# B&R Automation Studio project CombinedLinenSoiledA9KAN (part 2)

#### picu.ab
```automation-basic
PROGRAM _CYCLIC

;Sequence 24 - Primary Incline Conveyor 1 D[900 + mySeq]

;Note - Not a real sequence and not shown

;-----------------------------------------
;Revision 1.00 17/04/2007 D.J. First Issue
;-----------------------------------------

mySeq = 31
myIO = 172
myX20IO	= 23
myBufferBag = 841
myRelLine	= 65
myLine = 82 ; Line used to track bags
myZone	= 4

myLastBag = Line[myLine].LastBag
myFirstBag = Line[myLine].FirstBag
myRelBag = Line[myRelLine].LastBag

I_PaddleInPosition		= X[myIO].X01
I_BagReleasedSep		= X[myIO].X02
I_BagAtSep              = X[myIO].X03
I_ArriveIncline			= X[myIO].X04

O_RunMotor 				= FALSE
O_OpenSeparator			= FALSE

Alarm[mySeq].Name 	= 0
Alarm[mySeq].Bag	= myFirstBag
Alarm[mySeq].Beacon	= TRUE
Alarm[mySeq].Extra	= 0
Alarm[mySeq].Time	= 3000

;Setup Sequence
;-----------------------
STEP = D[900 + mySeq]
;Setup Pulse contact
PLS = (STEP <> LASTSTEP)
LASTSTEP = STEP

;If no bags on the buffers then stop the motor
NoBags = (Bag[myBufferBag].Cat = 0) AND (Bag[myFirstBag].Cat = 0)
TON_10ms(NoBags,10,StopIncline,StopInclineET)

O_RunMotor = (Line[myRelLine].Clear AND NOT Line[myRelLine].TripFault AND NOT StopIncline AND NOT Std.HaltSysZone[myZone] AND (STEP <> 2) AND (STEP <> 0))
IF (STEP = 0) THEN

ENDIF

;Run Incline until paddle in position
TON_10ms(I_BagAtSep,250,SettledInSep,SettledInSepET)
TON_10ms((Bag[myBufferBag].Cat > 0) AND NOT Std.HaltSysZone[myZone],300,SettledAtSep,SettledAtSepET)
IF (STEP = 1) THEN
	IF (I_PaddleInPosition AND O_RunMotor AND SettledAtSep AND (Bag[myLastBag].Cat = 0) AND (Bag[myBufferBag].Cat > 0)) THEN
		D[900 + mySeq] = 2
	ENDIF
ENDIF

;Release Bag into incline
IF (STEP = 2) THEN
	IF SettledInSep THEN
		BagArrived = TRUE
	ENDIF
	O_OpenSeparator	= (Bag[myLastBag].Cat = 0) AND NOT BagArrived

	IF I_ArriveIncline THEN
		IF ((Bag[myBufferBag].Cat > 0) AND (Bag[myLastBag].Cat = 0)) THEN
			Bag[myLastBag] = Bag[myBufferBag]
			Bag[myBufferBag] = Bag[0]
		ENDIF
		D[900 + mySeq] = 3
	ENDIF
	IF (Bag[myLastBag].Cat > 0) THEN
		Alarm[mySeq].Name = almBagDataError
		Alarm[mySeq].Time = 0
		Alarm[mySeq].Bag = myLastBag
	ELSE IF (Bag[myBufferBag].Cat > 0) AND NOT I_BagAtSep THEN
		Alarm[mySeq].Name = almSwitchFault
		Alarm[mySeq].Bag = myBufferBag
	ELSE
		Alarm[mySeq].Name = almBagNotReleased
		Alarm[mySeq].Bag = myBufferBag
	ENDIF
ELSE
	BagArrived = FALSE
ENDIF

;Check not stpped on paddle
IF (STEP = 3) THEN
	IF NOT I_PaddleInPosition THEN
		D[900 + mySeq] = 1
	ENDIF
ENDIF

;Move data from incline..
IF Line[myRelLine].Trip AND (Bag[myFirstBag].Cat > 0) AND (Bag[myRelBag].Cat = 0)  THEN ; Trip includes debounce
	Bag[myRelBag] = Bag[myFirstBag]
	Bag[myFirstBag] = Bag[0]
ENDIF

;Alarms
TimerAlarm.IN 		= NOT PLS AND (Alarm[mySeq].Name > 0)
TimerAlarm.PT 		= Alarm[mySeq].Time
TimerAlarm FUB TON_10ms()
Alarm[mySeq].On 	= TimerAlarm.Q
Alarm[mySeq].ET 	= TimerAlarm.ET
Alarm[mySeq].Zone 	= myZone

Y[myX20IO].Y02 	= O_RunMotor
Y[myIO].Y06 	= O_OpenSeparator AND NOT OpenSep
END_PROGRAM
```

### Program Logical/Reference/32_picd3 (IEC) - *PICD3 Incline Down Full bags

#### picd.var
```iecst
VAR
	TransitWindowClosedET : TIME;
	TransitWindowClosed : BOOL;
	TimerAlarm : TON_10ms;
	StopInclineET : TIME;
	StopIncline : BOOL;
	STEP : UINT;
	SettledAtSepET : UDINT;
	SettledAtSep : BOOL;
	ReleasedToInclineET : TIME;
	ReleasedToIncline : BOOL;
END_VAR
VAR RETAIN
	PLS : BOOL;
END_VAR
VAR
	O_RunMotor : BOOL;
	O_OpenSeparator : BOOL;
	NoBags : BOOL;
	myZone : INT;
	myX20IO : UINT;
	mySeq : UINT;
	myRelLine : UINT;
	myRelBag : UINT;
	myLine : UINT;
	myLastBag : UINT;
	myIO : UINT;
	myFirstBag : UINT;
	myBufferBag : UINT;
END_VAR
VAR RETAIN
	LASTSTEP : UINT;
END_VAR
VAR
	I_TrolleyOutAtBott : BOOL;
	I_TrolleyOnIncline : BOOL;
	I_PaddleInPosition : BOOL;
	I_OutgoingFull : BOOL;
	I_BagInSep : BOOL;
	I_BagAtSep : BOOL;
	I_ArriveIncline : BOOL;
	BagReleasedSep : BOOL;
	BagReleased : BOOL;
	BagArriveIncline : BOOL;
	SettledInSep : BOOL;
	SettledInSepET : UDINT;
	BagArrived : BOOL;
END_VAR
```

#### picd.ab
```automation-basic
PROGRAM _CYCLIC

;Sequence 24 - Primary Incline Conveyor 1 D[900 + mySeq]

;Note - Not a real sequence and not shown

;-----------------------------------------
;Revision 1.00 17/04/2007 D.J. First Issue
;-----------------------------------------

mySeq = 32
myIO = 173
myX20IO	= 33
myBufferBag = 891
myRelLine	= 68
myLine = 83 ; Line used to track bags
myZone	= 1

myLastBag = Line[myLine].LastBag
myFirstBag = Line[myLine].FirstBag
myRelBag = Line[myRelLine].LastBag

I_PaddleInPosition		= X[myIO].X01
I_BagInSep				= X[myIO].X02
I_BagAtSep              = X[myIO].X03
I_ArriveIncline			= X[myIO].X04

O_RunMotor 				= FALSE
O_OpenSeparator			= FALSE

Alarm[mySeq].Name 	= 0
Alarm[mySeq].Bag	= myFirstBag
Alarm[mySeq].Beacon	= TRUE
Alarm[mySeq].Extra	= 0
Alarm[mySeq].Time	= 3000

;Setup Sequence
;-----------------------
STEP = D[900 + mySeq]
;Setup Pulse contact
PLS = (STEP <> LASTSTEP)
LASTSTEP = STEP

;If no bags on the buffers then stop the motor
;NoBags = (Bag[myBufferBag].Cat = 0) AND (Bag[myFirstBag].Cat = 0)
NoBags = (((Bag[myFirstBag].Cat = 0) OR ((STEP = 1) AND Bag[myBufferBag].Cat > 0))  AND ((STEP = 1) AND I_PaddleInPosition))
IF NoBags THEN
	StopIncline = TRUE
ELSE IF (STEP <> 1) THEN
	StopIncline = FALSE
ENDIF

O_RunMotor = (Line[myRelLine].Clear AND NOT Line[myRelLine].TripFault AND NOT Std.HaltSysZone[myZone] AND (STEP <> 2) AND (STEP <> 0))
IF (STEP = 0) THEN

ENDIF

;Run Incline until paddle in position
TON_10ms(I_BagAtSep,25,SettledAtSep,SettledAtSepET)	;75
IF (STEP = 1) THEN
	IF ((I_PaddleInPosition OR StopIncline) AND O_RunMotor AND SettledAtSep AND (Bag[myLastBag].Cat = 0) AND (Bag[myBufferBag].Cat > 0) AND NOT I_BagInSep) THEN
		D[900 + mySeq] = 2
	ENDIF
	IF I_BagInSep THEN
		Alarm[mySeq].Name = almSwitchFault
	ENDIF
ENDIF

;Release Bag into incline

TON_10ms(I_BagInSep,25,SettledInSep,SettledInSepET)	;150
IF (STEP = 2) THEN

	IF SettledInSep THEN
		BagArrived = TRUE
	ENDIF
	O_OpenSeparator	= (Bag[myLastBag].Cat = 0) AND NOT BagArrived
	IF I_ArriveIncline THEN
		IF ((Bag[myBufferBag].Cat > 0) AND (Bag[myLastBag].Cat = 0)) THEN
			Bag[myLastBag] = Bag[myBufferBag]
			Bag[myBufferBag] = Bag[0]
		ENDIF
		D[900 + mySeq] = 3
	ENDIF
	IF (Bag[myLastBag].Cat > 0) THEN
		Alarm[mySeq].Name = almBagDataError
		Alarm[mySeq].Time = 0
		Alarm[mySeq].Bag = myLastBag
	ELSE
		Alarm[mySeq].Name = almBagNotReleased
		Alarm[mySeq].Bag = myBufferBag
	ENDIF
ELSE
	BagArrived = FALSE
ENDIF

;Check not stpped on paddle
IF (STEP = 3) THEN
	IF NOT I_PaddleInPosition THEN
		D[900 + mySeq] = 1
	ENDIF
ENDIF

;Move data from incline..
IF Line[myRelLine].Trip AND (Bag[myFirstBag].Cat > 0) AND (Bag[myRelBag].Cat = 0)  THEN ; Trip includes debounce
	Bag[myRelBag] = Bag[myFirstBag]
	Bag[myFirstBag] = Bag[0]
ENDIF

;Alarms
TimerAlarm.IN 		= NOT PLS AND (Alarm[mySeq].Name > 0)
TimerAlarm.PT 		= Alarm[mySeq].Time
TimerAlarm FUB TON_10ms()
Alarm[mySeq].On 	= TimerAlarm.Q
Alarm[mySeq].ET 	= TimerAlarm.ET
Alarm[mySeq].Zone 	= myZone

Y[myX20IO].Y01 	= O_RunMotor AND NOT StopIncline
Y[myIO].Y06 	= O_OpenSeparator
END_PROGRAM
```

### Program Logical/Reference/33_picd4 (IEC) - *PICD4 Incline Down Full bags

#### picd.ab
```automation-basic
PROGRAM _CYCLIC

;Sequence 24 - Primary Incline Conveyor 1 D[900 + mySeq]

;Note - Not a real sequence and not shown

;-----------------------------------------
;Revision 1.00 17/04/2007 D.J. First Issue
;-----------------------------------------

mySeq = 33
myIC = 4
myIO = 174
myX20IO	= 33
myBufferBag = 907
myRelLine	= 69
myLine = 84 ; Line used to track bags
myZone	= 1

myLastBag = Line[myLine].LastBag
myFirstBag = Line[myLine].FirstBag
myRelBag = Line[myRelLine].LastBag

I_PaddleInPosition		= X[myIO].X01
I_BagInSep				= X[myIO].X02
I_BagAtSep              = X[myIO].X03
I_ArriveIncline			= X[myIO].X04

O_RunMotor 				= FALSE
O_OpenSeparator			= FALSE
Enable.IC[myIC]			= FALSE

Alarm[mySeq].Name 	= 0
Alarm[mySeq].Bag	= myFirstBag
Alarm[mySeq].Beacon	= TRUE
Alarm[mySeq].Extra	= 0
Alarm[mySeq].Time	= 3000

;Setup Sequence
;-----------------------
STEP = D[900 + mySeq]
;Setup Pulse contact
PLS = (STEP <> LASTSTEP)
LASTSTEP = STEP

;If no bags on the buffers then stop the motor
NoBags = (((Bag[myFirstBag].Cat = 0) OR ((STEP = 1) AND Bag[myBufferBag].Cat > 0))  AND ((STEP = 1) AND I_PaddleInPosition))
IF NoBags THEN
	StopIncline = TRUE
ELSE IF (STEP <> 1) THEN
	StopIncline = FALSE
ENDIF

O_RunMotor = (Line[myRelLine].Clear AND NOT Line[myRelLine].TripFault AND NOT Std.HaltSysZone[myZone] AND (STEP <> 2) AND (STEP <> 0))
IF (STEP = 0) THEN

ENDIF

;Run Incline until paddle in position
TON_10ms(I_BagAtSep,25,SettledAtSep,SettledAtSepET)	;75
IF (STEP = 1) THEN
	IF ((I_PaddleInPosition OR StopIncline) AND O_RunMotor AND SettledAtSep AND (Bag[myLastBag].Cat = 0) AND (Bag[myBufferBag].Cat > 0) AND NOT I_BagInSep) THEN
		D[900 + mySeq] = 2
	ENDIF
	IF I_BagInSep THEN
		Alarm[mySeq].Name = almSwitchFault
	ENDIF
ENDIF

;Release Bag into incline

TON_10ms(I_BagInSep,150,SettledInSep,SettledInSepET)
IF (STEP = 2) THEN
	IF SettledInSep THEN
		BagArrived = TRUE
	ENDIF
	O_OpenSeparator	= (Bag[myLastBag].Cat = 0) AND NOT BagArrived
	IF I_ArriveIncline THEN
		IF ((Bag[myBufferBag].Cat > 0) AND (Bag[myLastBag].Cat = 0)) THEN
			Bag[myLastBag] = Bag[myBufferBag]
			Bag[myBufferBag] = Bag[0]
		ENDIF
		D[900 + mySeq] = 3
	ENDIF
	IF (Bag[myLastBag].Cat > 0) THEN
		Alarm[mySeq].Name = almBagDataError
		Alarm[mySeq].Time = 0
		Alarm[mySeq].Bag = myLastBag
	ELSE
		Alarm[mySeq].Name = almBagNotReleased
		Alarm[mySeq].Bag = myBufferBag
	ENDIF
ELSE
	BagArrived = FALSE
ENDIF

;Check not stpped on paddle
IF (STEP = 3) THEN
	IF NOT I_PaddleInPosition THEN
		D[900 + mySeq] = 1
	ENDIF
ENDIF

;Move data from incline..
IF Line[myRelLine].Trip AND (Bag[myFirstBag].Cat > 0) AND (Bag[myRelBag].Cat = 0)  THEN ; Trip includes debounce
	Bag[myRelBag] = Bag[myFirstBag]
	Bag[myFirstBag] = Bag[0]
ENDIF

;Alarms
TimerAlarm.IN 		= NOT PLS AND (Alarm[mySeq].Name > 0)
TimerAlarm.PT 		= Alarm[mySeq].Time
TimerAlarm FUB TON_10ms()
Alarm[mySeq].On 	= TimerAlarm.Q
Alarm[mySeq].ET 	= TimerAlarm.ET
Alarm[mySeq].Zone 	= myZone
Y[myX20IO].Y02 	= O_RunMotor AND NOT StopIncline
Y[myIO].Y06 	= O_OpenSeparator
END_PROGRAM
```

### Program Logical/Reference/35_picu6 (IEC) - *PICU6 Incline up Empty trolleys - Special not outgoing buffer

#### picu.var
```iecst
VAR RETAIN
	STEP : UINT;
	PLS : BOOL;
	LASTSTEP : UINT;
END_VAR
VAR
	O_RunMotor : BOOL;
	I_OutgoingFull : BOOL;
	O_OpenSeparator : BOOL;
	ReleasedToIncline : BOOL;
	ReleasedToInclineET : TIME;
	OutgoingFull : BOOL;
	OutgoingFullET : TIME;
	NoBags : BOOL;
	StopInclineET : TIME;
	StopIncline : BOOL;
	I_PaddleInPosition : BOOL;
	BagArriveIncline : BOOL;
	I_ArriveIncline : BOOL;
	TransitWindowClosedET : TIME;
	TransitWindowClosed : BOOL;
	BagReleasedSep : BOOL;
	I_BagAtSep : BOOL;
	I_LoadingInPosition : BOOL;
	TrackInPosET : TIME;
	TrackInPos : BOOL;
	mySeq : UINT;
	I_BagArriveIncline : BOOL;
	myIO : UINT;
	I_BagAtTopIncline : BOOL;
	I_BagReleased : BOOL;
	myIC : UINT;
	SettledSep : BOOL;
	SettledSepET : UDINT;
	myZone : INT;
	I_BagInSep : BOOL;
	SettledInSep : BOOL;
	SettledInSepET : UDINT;
	BagInSep : BOOL;
END_VAR
```

#### picu.ab
```automation-basic
PROGRAM _CYCLIC
	(* cyclic program *)

;Sequence 30 - Primary Incline Conveyor 4 D[900 + mySeq]
;Special incline - Only use 1 bag at time to store as buffer.
;-----------------------------------------
;Revision 1.00 17/04/2007 D.J. First Issue
;-----------------------------------------
mySeq 	= 35
myIO	= 176
myIC 	= 6
myZone	= 0

I_PaddleInPosition		= X[myIO].X01
I_BagAtSep              = X[myIO].X03
I_BagArriveIncline		= X[myIO].X04
I_BagInSep				= X[myIO].X02
I_BagReleased			= X[myIO].X05

O_RunMotor 				= FALSE
O_OpenSeparator			= FALSE
RequestRel.IC[myIC]		= FALSE

;Setup Sequence
;-----------------------
STEP = D[900 + mySeq]
;Setup Pulse contact
PLS = (STEP <> LASTSTEP)
LASTSTEP = STEP

IF (STEP = 0) THEN
;	D[900 + mySeq] = 1
ENDIF

;Run Incline until paddle in position
IF (STEP = 1) THEN
	O_RunMotor = TRUE
	IF I_PaddleInPosition AND NOT I_BagAtTopIncline THEN
		D[900 + mySeq] = 2
	ELSE IF I_BagAtTopIncline THEN
		Alarm[mySeq].Name = almSwitchFault
	ENDIF
ENDIF

;Step 2 wait for trolley at sep
TON_10ms(I_BagAtSep,200,SettledSep,SettledSepET)
	IF (STEP = 2) THEN
		IF SettledSep THEN
		D[900 + mySeq] = 3
	ENDIF
ENDIF

;Open Separator 1.5 seconds
TON_10ms(I_BagInSep,150,SettledInSep,SettledInSepET)
IF (STEP = 3) THEN
	IF SettledInSep THEN
		BagInSep = TRUE
	ENDIF
	O_OpenSeparator = NOT BagInSep
	IF I_BagArriveIncline THEN
		D[900 + mySeq] = 4
	ENDIF
	IF NOT Std.HaltSysZone[myZone] THEN
		Alarm[mySeq].Name = almBagNotArrived
	ENDIF
ELSE
	BagInSep = FALSE
ENDIF

;Step 4 Run incline until trolley is at the top
IF (STEP = 4) THEN
;	O_RunMotor = NOT EnableRel.IC[myIC]
;	IF I_BagAtTopIncline THEN
	IF NOT EnableRel.IC[myIC] THEN
		D[900 + mySeq] = 5
	ENDIF
;	ENDIF
;	IF EnableRel.IC[myIC] THEN
;		Alarm[mySeq].Name = almGeneralSequence
;	ENDIF
ENDIF

;Step 5 RequestRel
IF (STEP = 5) THEN
	RequestRel.IC[myIC] = NOT I_BagReleased
	IF EnableRel.IC[myIC] THEN
		D[900 + mySeq] = 6
	ENDIF
	IF  I_BagReleased AND NOT Std.HaltSysZone[myZone] THEN
		Alarm[mySeq].Name = almSwitchFault
	ENDIF
ENDIF

;Step 6 Run To Release trolley
IF (STEP = 6) THEN
	O_RunMotor = TRUE
	IF (I_BagReleased OR NOT EnableRel.IC[myIC]) THEN
		D[900 + mySeq] = 7
	ENDIF

ENDIF

;Check not stpped on paddle
IF (STEP = 7) THEN
	O_RunMotor = TRUE
	IF NOT I_PaddleInPosition THEN
		D[900 + mySeq] = 1
	ENDIF
ENDIF

Y[34].Y01		= O_RunMotor
Y[myIO].Y06 	= O_OpenSeparator
END_PROGRAM
```

### Program Logical/Reference/37_picu8 (IEC) - *PICU8 Incline up Empty trolleys

#### picu.ab
```automation-basic
PROGRAM _CYCLIC
	(* cyclic program *)

;Sequence 30 - Primary Incline Conveyor 4 D[900 + mySeq]

;-----------------------------------------
;Revision 1.00 17/04/2007 D.J. First Issue
;-----------------------------------------
mySeq 	= 37
myIO	= 178
myZone	= 0

I_PaddleInPosition		= X[myIO].X01
I_BagAtSep              = X[myIO].X03
I_BagArriveIncline		= X[myIO].X04
I_OutgoingFull			= X[myIO].X05

O_RunMotor 				= FALSE
O_OpenSeparator			= FALSE

;Setup Sequence
;-----------------------
STEP = D[900 + mySeq]
;Setup Pulse contact
PLS = (STEP <> LASTSTEP)
LASTSTEP = STEP

;If no bags on the buffers then stop the motor
NoBags = (STEP = 1) AND NOT I_BagAtSep
TON_10ms(NoBags,750,StopIncline,StopInclineET)
TON_10ms(I_OutgoingFull,100,OutgoingFull,OutgoingFullET)

O_RunMotor = (NOT OutgoingFull AND NOT StopIncline AND NOT Std.HaltSysZone[myZone] AND (STEP <> 0) AND (STEP <> 2)); AND (STEP <> 2))

IF (STEP = 0) THEN

ENDIF

;Run Incline until paddle in position
IF (STEP = 1) THEN
	IF (I_PaddleInPosition AND I_BagAtSep AND O_RunMotor) THEN
		D[900 + mySeq] = 2
	ENDIF
ENDIF

;Open Separator 1.5 seconds
;Allow 3 sec for trolley to be detected releasing from separator
TON_10ms((STEP = 2),150,ReleasedToIncline,ReleasedToInclineET)
TON_10ms(ReleasedToIncline,550,TransitWindowClosed,TransitWindowClosedET)
IF (STEP = 2) THEN
	O_OpenSeparator	= NOT ReleasedToIncline
	IF I_BagArriveIncline OR TransitWindowClosed THEN
		D[900 + mySeq] = 3
	ENDIF
	ELSE
	ReleasedToIncline = FALSE
ENDIF

;Check not stpped on paddle
IF (STEP = 3) THEN
	IF NOT I_PaddleInPosition THEN
		D[900 + mySeq] = 1
	ENDIF
ENDIF

Y[34].Y03 		= O_RunMotor
Y[myIO].Y06 	= O_OpenSeparator
END_PROGRAM
```

### Program Logical/Reference/40_picu11 (IEC) - *PICU11 Incline up Empty trolleys

#### picu.ab
```automation-basic
PROGRAM _CYCLIC
	(* cyclic program *)

;Sequence 30 - Primary Incline Conveyor 4 D[900 + mySeq]

;-----------------------------------------
;Revision 1.00 17/04/2007 D.J. First Issue
;-----------------------------------------
mySeq 	= 40
myIO	= 181
myZone	= 1

I_PaddleInPosition		= X[myIO].X01
I_BagAtSep              = X[myIO].X03
I_BagArriveIncline		= X[myIO].X04
I_OutgoingFull			= X[myIO].X05

O_RunMotor 				= FALSE
O_OpenSeparator			= FALSE

;Setup Sequence
;-----------------------
STEP = D[900 + mySeq]
;Setup Pulse contact
PLS = (STEP <> LASTSTEP)
LASTSTEP = STEP

;If no bags on the buffers then stop the motor
NoBags = (STEP = 1) AND NOT I_BagAtSep
TON_10ms(NoBags,3500,StopIncline,StopInclineET)
TON_10ms(I_OutgoingFull,100,OutgoingFull,OutgoingFullET)

O_RunMotor = (NOT OutgoingFull AND NOT StopIncline AND NOT Std.HaltSysZone[myZone] AND (STEP <> 0) AND (STEP <> 2))

IF (STEP = 0) THEN
	D[900 + mySeq] = 1
ENDIF

;Run Incline until paddle in position
IF (STEP = 1) THEN
	IF (I_PaddleInPosition AND I_BagAtSep AND O_RunMotor) THEN
		D[900 + mySeq] = 2
	ENDIF
ENDIF

;Open Separator 1.5 seconds
;Allow 3 sec for trolley to be detected releasing from separator
TON_10ms((STEP = 2),150,ReleasedToIncline,ReleasedToInclineET)
TON_10ms(ReleasedToIncline,550,TransitWindowClosed,TransitWindowClosedET)
IF (STEP = 2) THEN
	O_OpenSeparator	= NOT ReleasedToIncline
	IF TransitWindowClosed OR I_BagArriveIncline THEN
		D[900 + mySeq] = 3
	ENDIF
	ELSE
	ReleasedToIncline = FALSE
ENDIF

;Check not stpped on paddle
IF (STEP = 3) THEN
	IF NOT I_PaddleInPosition THEN
		D[900 + mySeq] = 1
	ENDIF
ENDIF

Y[33].Y04 		= O_RunMotor
Y[myIO].Y06 	= O_OpenSeparator
END_PROGRAM
```

### Program Logical/Reference/41_picd12 (IEC, version 1.00.0) - *PICU12 Incline down Empty trolleys

#### picu.ab
```automation-basic
PROGRAM _CYCLIC
	(* cyclic program *)

;Sequence 30 - Primary Incline Conveyor 4 D[900 + mySeq]

;-----------------------------------------
;Revision 1.00 17/04/2007 D.J. First Issue
;-----------------------------------------
mySeq 	= 41
myIO	= 182
myZone	= 0

I_PaddleInPosition		= X[myIO].X01
I_BagAtSep              = X[myIO].X03
I_BagArriveIncline		= X[myIO].X04
I_OutgoingFull			= X[myIO].X05

O_RunMotor 				= FALSE
O_OpenSeparator			= FALSE

;Setup Sequence
;-----------------------
STEP = D[900 + mySeq]
;Setup Pulse contact
PLS = (STEP <> LASTSTEP)
LASTSTEP = STEP

;If no bags on the buffers then stop the motor
NoBags = (STEP = 1) AND NOT I_BagAtSep
TON_10ms(NoBags,6000,StopIncline,StopInclineET)
TON_10ms(I_OutgoingFull,100,OutgoingFull,OutgoingFullET)

O_RunMotor = (NOT OutgoingFull AND NOT StopIncline AND NOT Std.HaltSysZone[myZone] AND (STEP <> 2))

IF (STEP = 0) THEN
	D[900 + mySeq] = 1
ENDIF

;Run Incline until paddle in position
IF (STEP = 1) THEN
	IF (I_PaddleInPosition AND I_BagAtSep AND O_RunMotor) THEN
		D[900 + mySeq] = 2
	ENDIF
ENDIF

;Open Separator 1.5 seconds
;Allow 3 sec for trolley to be detected releasing from separator
TON_10ms((STEP = 2),150,ReleasedToIncline,ReleasedToInclineET)
TON_10ms(ReleasedToIncline,550,TransitWindowClosed,TransitWindowClosedET)
IF (STEP = 2) THEN
	O_OpenSeparator	= NOT ReleasedToIncline
	IF TransitWindowClosed OR I_BagArriveIncline THEN
		D[900 + mySeq] = 3
	ENDIF
	ELSE
	ReleasedToIncline = FALSE
ENDIF

;Check not stpped on paddle
IF (STEP = 3) THEN
	IF NOT I_PaddleInPosition THEN
		D[900 + mySeq] = 1
	ENDIF
ENDIF

Y[23].Y03 		= O_RunMotor
Y[myIO].Y06 	= O_OpenSeparator
END_PROGRAM
```

### Program Logical/Reference/43_picd14 (IEC) - *PICU14 Incline down Empty trolleys

#### picu.ab
```automation-basic
PROGRAM _CYCLIC
	(* cyclic program *)

;Sequence 30 - Primary Incline Conveyor 4 D[900 + mySeq]

;-----------------------------------------
;Revision 1.00 17/04/2007 D.J. First Issue
;-----------------------------------------
mySeq 	= 43
myIO	= 184
myZone	= 3

I_PaddleInPosition		= X[myIO].X01
I_BagAtSep              = X[myIO].X03
I_BagArriveIncline		= X[myIO].X04
I_OutgoingFull			= X[myIO].X05

O_RunMotor 				= FALSE
O_OpenSeparator			= FALSE

;Setup Sequence
;-----------------------
STEP = D[900 + mySeq]
;Setup Pulse contact
PLS = (STEP <> LASTSTEP)
LASTSTEP = STEP

;If no bags on the buffers then stop the motor
NoBags = (STEP = 1) AND NOT I_BagAtSep
TON_10ms(NoBags,2000,StopIncline,StopInclineET)
TON_10ms(I_OutgoingFull,100,OutgoingFull,OutgoingFullET)

O_RunMotor = (NOT OutgoingFull AND NOT StopIncline AND NOT Std.HaltSysZone[myZone] AND (STEP <> 2))

IF (STEP = 0) THEN
	D[900 + mySeq] = 1
ENDIF

;Run Incline until paddle in position
IF (STEP = 1) THEN
	IF (I_PaddleInPosition AND I_BagAtSep AND O_RunMotor) THEN
		D[900 + mySeq] = 2
	ENDIF
ENDIF

;Open Separator 1.5 seconds
;Allow 3 sec for trolley to be detected releasing from separator
TON_10ms((STEP = 2),150,ReleasedToIncline,ReleasedToInclineET)
TON_10ms(ReleasedToIncline,550,TransitWindowClosed,TransitWindowClosedET)
IF (STEP = 2) THEN
	O_OpenSeparator	= NOT ReleasedToIncline
	IF TransitWindowClosed OR I_BagArriveIncline THEN
		D[900 + mySeq] = 3
	ENDIF
	ELSE
	ReleasedToIncline = FALSE
ENDIF

;Check not stpped on paddle
IF (STEP = 3) THEN
	IF NOT I_PaddleInPosition THEN
		D[900 + mySeq] = 1
	ENDIF
ENDIF

Y[23].Y05 		= O_RunMotor
Y[myIO].Y06 	= O_OpenSeparator
END_PROGRAM
```

### Program Logical/Reference/44_picd15 (IEC) - *PICU15 Incline down Empty trolleys

#### picu.var
```iecst
VAR RETAIN
	STEP : UINT;
	PLS : BOOL;
	LASTSTEP : UINT;
	O_RunMotor : BOOL;
	I_OutgoingFull : BOOL;
	O_OpenSeparator : BOOL;
	ReleasedToIncline : BOOL;
	ReleasedToInclineET : TIME;
	OutgoingFull : BOOL;
	OutgoingFullET : TIME;
	NoBags : BOOL;
	StopInclineET : TIME;
	StopIncline : BOOL;
END_VAR
VAR
	I_PaddleInPosition : BOOL;
	BagArriveIncline : BOOL;
	I_ArriveIncline : BOOL;
	TransitWindowClosedET : TIME;
	TransitWindowClosed : BOOL;
	BagReleasedSep : BOOL;
	I_BagAtSep : BOOL;
	I_LoadingInPosition : BOOL;
	TrackInPosET : TIME;
	TrackInPos : BOOL;
	mySeq : UINT;
	I_BagArriveIncline : BOOL;
	myIO : UINT;
	myZone : INT;
END_VAR
```

### Program Logical/Reference/45_picu16 (IEC) - *PICU16 Incline up Empty trolleys

#### picu.ab
```automation-basic
PROGRAM _CYCLIC
	(* cyclic program *)

;Sequence 30 - Primary Incline Conveyor 4 D[900 + mySeq]

;-----------------------------------------
;Revision 1.00 17/04/2007 D.J. First Issue
;-----------------------------------------
mySeq 	= 45
myIO	= 186
myZone	= 0

I_PaddleInPosition		= X[myIO].X01
I_BagAtSep              = X[myIO].X03
I_BagArriveIncline		= X[myIO].X04
I_OutgoingFull			= X[myIO].X05

O_RunMotor 				= FALSE
O_OpenSeparator			= FALSE

;Setup Sequence
;-----------------------
STEP = D[900 + mySeq]
;Setup Pulse contact
PLS = (STEP <> LASTSTEP)
LASTSTEP = STEP

;If no bags on the buffers then stop the motor
NoBags = (STEP = 1) AND NOT I_BagAtSep
TON_10ms(NoBags,2000,StopIncline,StopInclineET)
TON_10ms(I_OutgoingFull,100,OutgoingFull,OutgoingFullET)

O_RunMotor = (NOT OutgoingFull AND NOT StopIncline AND NOT Std.HaltSysZone[myZone] AND (STEP <> 0) AND (STEP <> 2)); AND (STEP <> 2))

IF (STEP = 0) THEN
;	D[900 + mySeq] = 1
ENDIF

;Run Incline until paddle in position
IF (STEP = 1) THEN
	IF (I_PaddleInPosition AND I_BagAtSep AND O_RunMotor) THEN
		D[900 + mySeq] = 2
	ENDIF
ENDIF

;Open Separator 1.5 seconds
;Allow 3 sec for trolley to be detected releasing from separator
TON_10ms((STEP = 2),150,ReleasedToIncline,ReleasedToInclineET)
TON_10ms(ReleasedToIncline,550,TransitWindowClosed,TransitWindowClosedET)
IF (STEP = 2) THEN
	O_OpenSeparator	= NOT ReleasedToIncline
	IF I_BagArriveIncline OR TransitWindowClosed THEN
		D[900 + mySeq] = 3
	ENDIF
	ELSE
	ReleasedToIncline = FALSE
ENDIF

;Check not stpped on paddle
IF (STEP = 3) THEN
	IF NOT I_PaddleInPosition THEN
		D[900 + mySeq] = 1
	ENDIF
ENDIF

Y[34].Y06		= O_RunMotor
Y[myIO].Y06 	= O_OpenSeparator
END_PROGRAM
```

### Program Logical/Reference/46_picu17 (IEC) - *PICU17 Incline up Empty trolleys

#### picu.ab
```automation-basic
PROGRAM _CYCLIC
	(* cyclic program *)

;Sequence 30 - Primary Incline Conveyor 4 D[900 + mySeq]

;-----------------------------------------
;Revision 1.00 17/04/2007 D.J. First Issue
;-----------------------------------------
mySeq 	= 46
myIO	= 187
myZone	= 0

I_PaddleInPosition		= X[myIO].X01
I_BagAtSep              = X[myIO].X03
I_BagArriveIncline		= X[myIO].X04
I_OutgoingFull			= X[myIO].X05

O_RunMotor 				= FALSE
O_OpenSeparator			= FALSE

;Setup Sequence
;-----------------------
STEP = D[900 + mySeq]
;Setup Pulse contact
PLS = (STEP <> LASTSTEP)
LASTSTEP = STEP

;If no bags on the buffers then stop the motor
NoBags = (STEP = 1) AND NOT I_BagAtSep
TON_10ms(NoBags,2000,StopIncline,StopInclineET)
TON_10ms(I_OutgoingFull,100,OutgoingFull,OutgoingFullET)

O_RunMotor = (NOT OutgoingFull AND NOT StopIncline AND NOT Std.HaltSysZone[myZone] AND (STEP <> 0) AND (STEP <> 2)); AND (STEP <> 2))

IF (STEP = 0) THEN
;	D[900 + mySeq] = 1
ENDIF

;Run Incline until paddle in position
IF (STEP = 1) THEN
	IF (I_PaddleInPosition AND I_BagAtSep AND O_RunMotor) THEN
		D[900 + mySeq] = 2
	ENDIF
ENDIF

;Open Separator 1.5 seconds
;Allow 3 sec for trolley to be detected releasing from separator
TON_10ms((STEP = 2),150,ReleasedToIncline,ReleasedToInclineET)
TON_10ms(ReleasedToIncline,550,TransitWindowClosed,TransitWindowClosedET)
IF (STEP = 2) THEN
	O_OpenSeparator	= NOT ReleasedToIncline
	IF I_BagArriveIncline OR TransitWindowClosed THEN
		D[900 + mySeq] = 3
	ENDIF
	ELSE
	ReleasedToIncline = FALSE
ENDIF

;Check not stpped on paddle
IF (STEP = 3) THEN
	IF NOT I_PaddleInPosition THEN
		D[900 + mySeq] = 1
	ENDIF
ENDIF

Y[34].Y07		= O_RunMotor
Y[myIO].Y06 	= O_OpenSeparator
END_PROGRAM
```

### Program Logical/Reference/48_49_fbppr (IEC) - *Full bag pressure reliefs buffers before PUPs

#### fb_pr.ab
```automation-basic
;--------------------------------------------
;Sequence 0 - XXX0  D[900 + mySeq]
;--------------------------------------------

PROGRAM _INIT
(* init program *)
END_PROGRAM

PROGRAM _CYCLIC

;Inputs
mySeq				= 48 - 1	;Sequence number - 1 for arrays to work
myZone				= 0
;Index relates to line on storage,,
I_BagAtPR[1]		= X[125].X01
I_BagAtPR[2]		= X[129].X01

I_BagInSep[1]	= X[125].X03
I_BagInSep[2]	= X[129].X03

myLine[1]			= 76
myLine[2]			= 75
myOutLine[1]		= 74
myOutLine[2]		= 73

LOOP x = 1 TO Dec_C_MaxPressureReliefs DO
	IF TestIndex > 0 THEN
		n = TestIndex
	ELSE
		n = x
	ENDIF
	O_OpenStop[n] = FALSE

	Alarm[mySeq + n].Name 	= 0
	Alarm[mySeq + n].Bag	= 0
	Alarm[mySeq + n].Beacon	= TRUE
	Alarm[mySeq + n].Extra	= 0
	Alarm[mySeq + n].Time	= 3000

	BagSettled[n].IN = I_BagAtPR[n]
	BagSettled[n].PT = 75
	BagSettled[n] FUB TON_10ms()

	SettledInSep[n].IN = I_BagInSep[n]
	SettledInSep[n].PT = 75
	SettledInSep[n] FUB TON_10ms()
	;Setup Sequence
	STEP = D[900 + mySeq + n]
	;Setup Pulse contact
	PLS[n] = (STEP <> LASTSTEP[n])
	LASTSTEP[n] = STEP

	;Set up local vars
	myBag = Line[myLine[n]].FirstBag
	myRelLine = myOutLine[n]
	myLastBag = Line[myRelLine].LastBag

	IF 	(STEP < 2) THEN
		BagReleased[n] = FALSE
	ELSE IF I_BagInSep[n] THEN
		BagReleased[n] = TRUE
	ENDIF
	;Sequence
	IF (STEP = 0) THEN
		;D[900 + mySeq + n -1] = 1
	ENDIF

	;Bag Settles at PR
	IF (STEP = 1) THEN
		IF (BagSettled[n].Q  AND (Bag[myBag].Cat > 0) AND  Line[myRelLine].Clear AND (Bag[myLastBag].Cat = 0)AND NOT Line[myRelLine].TripFault AND NOT Std.HaltSysZone[myZone])THEN
			ReleaseValid[n] = TRUE
		ENDIF
		O_OpenStop[n] = ReleaseValid[n]
		IF SettledInSep[n].Q THEN
			D[900 + mySeq + n] = 2
		ENDIF
		IF BagSettled[n].Q  AND (Bag[myBag].Cat = 0) THEN
			Alarm[mySeq + n].Name =  almSwitchFault
		ELSE IF O_OpenStop[n] AND NOT I_BagInSep[n] THEN
			Alarm[mySeq + n].Name =  almSwitchFault
		ELSE IF Line[myRelLine].TripFault THEN
			Alarm[mySeq + n].Name =  almSwitchFault
		ENDIF
	ELSE
		ReleaseValid[n] = FALSE
	ENDIF

	IF (STEP = 2) THEN
		;O_OpenStop[n] = TRUE
		IF Line[myRelLine].Trip THEN
			Bag[myLastBag] = Bag[myBag]
			Bag[myBag] = Bag[0]
			D[900 + mySeq + n] = 1
		ENDIF
		IF NOT Std.HaltSysZone[myZone] THEN
			Alarm[mySeq + n].Name = almBagNotReleased
		ENDIF
	ENDIF

	;Alarms
	TimerAlarm[n].IN 		= NOT PLS[n] AND (Alarm[mySeq + n].Name > 0)
	TimerAlarm[n].PT 		= Alarm[mySeq + n].Time
	TimerAlarm[n] FUB TON_10ms()
	Alarm[mySeq + n].On 	= TimerAlarm[n].Q
	Alarm[mySeq + n].ET 	= TimerAlarm[n].ET
	Alarm[mySeq + n].Zone 	= myZone
ENDLOOP

;-----------------------------------
;PLC Outputs - adjust to suit system
;-----------------------------------
Y[125].Y05 = O_OpenStop[1]
Y[129].Y05 = O_OpenStop[2]

END_PROGRAM
```

### Program Logical/Reference/50_fb_pr (IEC) - *Full bag pressure reliefs

#### fb_pr.var
```iecst
VAR CONSTANT
	Dec_C_MaxPressureReliefs : UINT := 1;
END_VAR
VAR RETAIN
	LASTSTEP : ARRAY[0..Dec_C_MaxPressureReliefs] OF UINT;
END_VAR
VAR
	PLS : ARRAY[0..Dec_C_MaxPressureReliefs] OF BOOL;
	STEP : UINT;
	TimerAlarm : ARRAY[0..Dec_C_MaxPressureReliefs] OF TON_10ms;
	mySeq : UINT;
	I_BagAtPR : ARRAY[0..Dec_C_MaxPressureReliefs] OF BOOL;
	n : INT;
	BagSettled : ARRAY[0..Dec_C_MaxPressureReliefs] OF TON_10ms;
	myRelLine : UINT;
	myLastBag : UINT;
	myBag : UINT;
	O_OpenStop : ARRAY[0..Dec_C_MaxPressureReliefs] OF BOOL;
	myZone : INT;
END_VAR
VAR RETAIN
	ReleaseValid : ARRAY[0..Dec_C_MaxPressureReliefs] OF BOOL;
END_VAR
VAR
	TON_10msReleaseValid : ARRAY[0..Dec_C_MaxPressureReliefs] OF TON_10ms;
	TimeOutTimer : ARRAY[0..Dec_C_MaxPressureReliefs] OF TON_10ms;
	DebugTimeOut_Counter : ARRAY[0..Dec_C_MaxPressureReliefs] OF UDINT;
END_VAR
```

#### fb_pr.ab
```automation-basic
;--------------------------------------------
;Sequence 0 - XXX0  D[900 + mySeq]
;--------------------------------------------

PROGRAM _INIT
(* init program *)
END_PROGRAM

PROGRAM _CYCLIC

;Inputs
mySeq				= 50	;Sequence number
myZone				= 4

;Index relates to line on storage,,
I_BagAtPR[1]		= X[211].X01

LOOP n = 1 TO Dec_C_MaxPressureReliefs DO

	O_OpenStop[n] = FALSE

	Alarm[mySeq + n].Name 	= 0
	Alarm[mySeq + n].Bag	= 0
	Alarm[mySeq + n].Beacon	= TRUE
	Alarm[mySeq + n].Extra	= 0
	Alarm[mySeq + n].Time	= 3000

	BagSettled[n].IN = I_BagAtPR[n]
	BagSettled[n].PT = 75
	BagSettled[n] FUB TON_10ms()

	TimeOutTimer[n].IN = (D[900 + mySeq + n] = 2)
	TimeOutTimer[n].PT = 6000
	TimeOutTimer[n] FUB TON_10ms()

	;Setup Sequence
	STEP = D[900 + mySeq + n]
	;Setup Pulse contact
	PLS[n] = (STEP <> LASTSTEP[n])
	LASTSTEP[n] = STEP

	;Set up local vars
	myBag = Line[n].FirstBag
	myRelLine = n + 20
	myLastBag = Line[myRelLine].LastBag

	;Sequence
	IF (STEP = 0) THEN
		D[900 + mySeq + n] = 1
	ENDIF
	TON_10msReleaseValid[n].IN = ((D[900 + mySeq + n] = 1) AND (Bag[myBag].Cat > 0) AND  Line[myRelLine].Clear AND (Bag[myLastBag].Cat = 0)AND NOT I_BagAtPR[n] AND NOT Line[myRelLine].TripFault AND NOT Std.HaltSysZone[myZone])
	TON_10msReleaseValid[n].PT = 450 ;Must be longer then Line full timer  + Travel time
	TON_10msReleaseValid[n] FUB TON_10ms()
	;Bag Settles at PR
	IF (STEP = 1) THEN
		IF TON_10msReleaseValid[n].Q THEN
			ReleaseValid[n] = TRUE
		ENDIF
		O_OpenStop[n] = ReleaseValid[n]
		IF BagSettled[n].Q THEN
			D[900 + mySeq + n] = 2
		ENDIF
		IF BagSettled[n].Q  AND (Bag[myBag].Cat = 0) THEN
			Alarm[mySeq + n].Name =  almSwitchFault
		ELSE IF Line[myRelLine].TripFault THEN
			Alarm[mySeq + n].Name =  almSwitchFault
		ENDIF
	ELSE
		ReleaseValid[n] = FALSE
	ENDIF

	IF (STEP = 2) THEN
		;O_OpenStop[n] = TRUE
		IF Line[myRelLine].Trip THEN ;OR Line[myRelLine].LongTrip THEN
			Bag[myLastBag] = Bag[myBag]
			Bag[myBag] = Bag[0]
			D[900 + mySeq + n] = 1
		ELSE IF TimeOutTimer[n].Q THEN
			INC DebugTimeOut_Counter[n]
			D[900 + mySeq + n] = 1
		ENDIF
		IF NOT Std.HaltSysZone[myZone] THEN
			Alarm[mySeq + n].Name = almBagNotReleased
		ENDIF
	ENDIF

	;Alarms
	TimerAlarm[n].IN 		= NOT PLS[n] AND (Alarm[mySeq + n].Name > 0)
	TimerAlarm[n].PT 		= Alarm[mySeq + n].Time
	TimerAlarm[n] FUB TON_10ms()
	Alarm[mySeq + n].On 	= TimerAlarm[n].Q
	Alarm[mySeq + n].ET 	= TimerAlarm[n].ET
	Alarm[mySeq + n].Zone 	= myZone
ENDLOOP

;-----------------------------------
;PLC Outputs - adjust to suit system
;-----------------------------------
Y[211].Y05 = O_OpenStop[1]
Y[211].Y06 = O_OpenStop[2]
Y[212].Y05 = O_OpenStop[3]
Y[212].Y06 = O_OpenStop[4]
Y[213].Y05 = O_OpenStop[5]
Y[213].Y06 = O_OpenStop[6]
Y[214].Y05 = O_OpenStop[7]
Y[214].Y06 = O_OpenStop[8]
Y[215].Y05 = O_OpenStop[9]
Y[215].Y06 = O_OpenStop[10]
Y[216].Y05 = O_OpenStop[11]
Y[216].Y06 = O_OpenStop[12]
Y[229].Y05 = O_OpenStop[15]

Y[217].Y05 = O_OpenStop[21]
Y[217].Y06 = O_OpenStop[22]
Y[218].Y05 = O_OpenStop[23]
Y[218].Y06 = O_OpenStop[24]
Y[219].Y05 = O_OpenStop[25]
Y[219].Y06 = O_OpenStop[26]
Y[220].Y05 = O_OpenStop[27]
Y[220].Y06 = O_OpenStop[28]
Y[221].Y05 = O_OpenStop[29]
Y[221].Y06 = O_OpenStop[30]
Y[222].Y05 = O_OpenStop[31]
Y[222].Y06 = O_OpenStop[32]
Y[231].Y06 = O_OpenStop[35]

END_PROGRAM
```

### Package Logical/Sequences - *GCS Primary 

### Package Logical/Sequences/10ms - 10ms Tasks

### Program Logical/Sequences/10ms/zzPrimSearch (IEC) - *Search for ongoing lines using SLAC looking at last bag in transit

#### zzPrimSearch.ab - Implementation code
```automation-basic
(********************************************************************
 * COPYRIGHT -- HP
 ********************************************************************
 * Program: zzPrimSearch
 * File: zzPrimSearch.ab
 * Author: treamsbottom
 * Created: May 09, 2014
 ********************************************************************
 * Implementation of program zzPrimSearch
 ********************************************************************)

PROGRAM _INIT

END_PROGRAM

PROGRAM _CYCLIC

;Find destination of primary bags using SLAC. As there are multiple Bags in transit before PPN use the last bag in transit for the calculation.

MaxBuffers 		= 1
MinLine			= 1
MaxLine			= 10
myStartStop		= 7700 // 7700 means 100 on tview
MaxDepth		= 17
myTransitLine	= 32; Ongoing line transfers multiple bags

OngoingEnabled = (D[4]>0)

BufferBagNum[1] = Line[16].FirstBag
//BufferBagNum[2] = Line[65].FirstBag

;Search only 1 buffer bag per scan/task
Buffer = Buffer + 1
IF Buffer > MaxBuffers THEN
	Buffer = 1
ENDIF
;Set Test Value for Monitoring
IF TestBuffer > 0 THEN
	Buffer = TestBuffer
ENDIF

BufferBag		= BufferBagNum[Buffer]
BufferSettled 	= TRUE
BufferPrg 		= Bag[BufferBag].Prg
BufferCat		= Bag[BufferBag].Cat
BufferCus		= Bag[BufferBag].Cus
BufferDst 		= Bag[BufferBag].Dst

IF (BufferSettled AND (BufferCat > 0) AND (BufferPrg > 0) AND (BufferPrg <= Std.MaxProg) AND OngoingEnabled) THEN

	;Manual Destination has been set?
	IF (BufferDst > 0) THEN
;		n = BufferDst
;
;		IF ((n >= MinLine) AND (n <= MaxLine) AND (Line[n].Space > 0) AND Line[n].Clear) THEN
;			Dest 	= n
;			Buff 	= Buffer
;
;		ELSE
;			Alarm[mySeq].Name 	= almDestinationNotValid
;			Alarm[mySeq].Bag	= BufferBag
;		ENDIF
;

	ELSE IF Std.AutoLineAllocation THEN ;/BufferDst > 0

		;Search Each Storage Area
		AreaChoice[1] = D[3000 + BufferPrg]
		AreaChoice[2] = D[3100 + BufferPrg]
		AreaChoice[3] = D[3200 + BufferPrg]
		AreaChoice[4] = D[3300 + BufferPrg]

		LOOP Area = 1 TO 4 DO
			Dest = 0

			AreaStartLine 	= D[250 + AreaChoice[Area]]
			AreaEndLine 	= D[270 + AreaChoice[Area]]
			AreaValid		= ((AreaStartLine > 0) AND (AreaEndLine > 0) AND (AreaEndLine >= AreaStartLine))
			IF AreaValid THEN

				;Search other buffers, as if destination has already been assigned for an empty a different line would be assigned due to BIT calc
				IF (Dest = 0) THEN
					LOOP n = 1 TO MaxBuffers DO
						IF (n <> Buffer) THEN ; Don't check self
							myBag = BufferBagNum[n]
							Match = (Bag[myBag].Prg = BufferPrg); AND (Bag[myBag].Cus = BufferCus)
							SearchDest = Bag[myBag].Dst
							myLineValid = ((SearchDest >= MinLine) AND (SearchDest <= MaxLine))
							myLineUsed	= (D[myStartStop + SearchDest] > 0) ;Start / Stop On
							IF (Match AND myLineValid AND myLineUsed AND (Line[SearchDest].SpaceBIT > 0) AND Line[SearchDest].Clear) THEN
								Dest = SearchDest
							ENDIF
						ENDIF
						EXITIF (Dest > 0)
					ENDLOOP
				ENDIF

				; Search ongoing transit buffer to find matching prg's; and customers later if requested
				IF (Dest = 0) THEN
					LOOP n = Line[myTransitLine].FirstBag TO Line[myTransitLine].LastBag DO
						Match = (Bag[n].Prg = BufferPrg); AND (Bag[n].Cus = BufferCus)
						SearchDest = Bag[n].Dst
						myLineValid = ((SearchDest >= MinLine) AND (SearchDest <= MaxLine))
						myLineUsed	= (D[myStartStop + SearchDest] > 0) ;Start / Stop On
						IF (Match AND myLineValid AND myLineUsed AND (Line[SearchDest].SpaceBIT > 0) AND Line[SearchDest].Clear) THEN
							Dest = SearchDest
						ENDIF
					EXITIF (Dest > 0)
					ENDLOOP
				ENDIF

				;Search for a line with the same program
					;---------------------------------------
				IF (Dest = 0) THEN
					LOOP myLine = AreaStartLine TO AreaEndLine DO
						myLineValid = ((myLine >= MinLine) AND (myLine <= MaxLine))
						myLineUsed	= (D[myStartStop + myLine] > 0) ;Start / Stop On
						IF myLineValid AND myLineUsed THEN
							n 			= myLine
							SearchBag[0] 	= (Line[n].LastBag - Line[n].Space)
;							SearchBag[1]    = (Line[n + 20].LastBag - Line[n + 20].Space)
;							SearchBag[2]    = (Line[n + 40].LastBag - Line[n + 40].Space)
							Condtion[1] 	= ((SearchBag[0] >= Line[n].FirstBag) AND (Bag[SearchBag[0]].Prg = BufferPrg))
;							Condtion[2] 	= ((SearchBag[1] >= Line[n + 20].FirstBag) AND (Bag[SearchBag[1]].Prg = BufferPrg))
;							Condtion[3] 	= ((SearchBag[2] >= Line[n + 40].FirstBag) AND (Bag[SearchBag[2]].Prg = BufferPrg))
							Match = (Condtion[1] OR Condtion[2] OR Condtion[3])
							IF (Match  AND (Line[n].SpaceBIT > 0) AND Line[n].Clear) THEN
								;Found line with a matching program
								Dest 	= n
							ENDIF ;/SearchBag[0]
						ENDIF ;/myLineValid
						EXITIF (Dest <> 0)
					ENDLOOP ;/myLine loop
				ENDIF
				;Search for an empty line
				;------------------------
				IF (Dest = 0) THEN
					LOOP myLine = AreaStartLine TO AreaEndLine DO
						myLineValid = ((myLine >= MinLine) AND (myLine <= MaxLine))
						myLineUsed	= (D[myStartStop + myLine] > 0) ;Start / Stop On
						IF myLineValid AND myLineUsed THEN
							n 			= myLine
							SearchBag[0] 	= (Line[n].FirstBag)
;							SearchBag[1]    = (Line[n + 20].LastBag - Line[n + 20].Space)
;							SearchBag[2]    = (Line[n + 40].LastBag - Line[n + 40].Space)
							Match = (Bag[SearchBag[0]].Prg = 0)// AND (Bag[SearchBag[1]].Prg = 0) AND (Bag[SearchBag[2]].Prg = 0))
							IF (Match AND (Line[n].SpaceBIT = Line[n].Space ) AND Line[n].Clear) THEN
								;Found line with a matching program
								Dest 	= n
							ENDIF ;/SearchBag[0]
						ENDIF ;/myLineValid
						EXITIF (Dest <> 0)
					ENDLOOP ;/myLine loop
				ENDIF ;/Dest = 0

;				Search for a line that already contains a bag with the same Program starting at the back
;				----------------------------------------------------------------------------------------
				IF (Dest = 0) THEN
					LOOP myDepth = (MaxDepth - 2) DOWNTO 0 DO ;Don't search the last bag as the line would already be full!!
						LOOP myLine = AreaStartLine TO AreaEndLine DO
							//LOOP LineIndex = 0 TO 2 DO
								myLineValid = ((myLine >= MinLine) AND (myLine <= MaxLine))
								myLineUsed	= (D[myStartStop + myLine] > 0) ;Start / Stop On
								IF myLineValid AND myLineUsed THEN
									n 			= myLine
									SearchBag[0] 	= (Line[n].FirstBag + myDepth)
									IF ((Bag[SearchBag[0]].Prg = BufferPrg) AND (Line[n].SpaceBIT > 0) AND Line[n].Clear) THEN
										;Found line with a matching program
										FoundDepth 	= myDepth
										Dest 		= myLine
									ENDIF ;/SearchBag[0]
								ENDIF ;/myLineValid
								//EXITIF (Dest <> 0)
							//ENDLOOP
							EXITIF (Dest <> 0)
						ENDLOOP ;/myLine loop
						EXITIF (Dest <> 0)
					ENDLOOP ;/myDepgh
				ENDIF ;/Dest = 0

				;Search for a line that already contains a bag with the same customer starting at the back
				;----------------------------------------------------------------------------------------
				IF (Dest = 0) THEN
					LOOP myDepth = (MaxDepth - 2) DOWNTO 0 DO ;Don't search the last bag as the line would already be full!!
						LOOP myLine = AreaStartLine TO AreaEndLine DO
							//LOOP LineIndex = 0 TO 2 DO
								myLineValid = ((myLine >= MinLine) AND (myLine <= MaxLine))
								myLineUsed	= (D[myStartStop + myLine] > 0) ;Start / Stop On
								IF myLineValid AND myLineUsed THEN
									n 			= myLine
									SearchBag[0] 	= (Line[n].FirstBag + myDepth)
									IF ((Bag[SearchBag[0]].Cus  = BufferCus) AND (Line[n].SpaceBIT > 0) AND Line[n].Clear) THEN
										;Found line with a matching program
										FoundDepth 	= myDepth
										Dest 		= myLine
									ENDIF ;/SearchBag[0]
								ENDIF ;/myLineValid
							//EXITIF (Dest <> 0)
							//ENDLOOP
						EXITIF (Dest <> 0)
						ENDLOOP ;/myLine loop
						EXITIF (Dest <> 0)
					ENDLOOP ;/myDepgh
				ENDIF ;/Dest = 0

				;Search for line with the most space
				;-----------------------------------
				IF (Dest = 0) THEN
					mySpace = 0
					myFound	= 0
					LOOP myLine = AreaStartLine TO AreaEndLine DO
						myLineValid = ((myLine >= MinLine) AND (myLine <= MaxLine))
						myLineUsed	= (D[myStartStop + myLine] > 0) ;Start / Stop On
						IF myLineValid AND myLineUsed THEN
							n 			= myLine
							SearchBag[0] 	= (Line[n].LastBag)
							LineSpace = Line[n].SpaceBIT
							IF ((Bag[SearchBag[0]].Prg = 0) AND (LineSpace > mySpace) AND (Line[n].SpaceBIT > 0)  AND Line[n].Clear) THEN
								;Found line with a matching program
								myFound	= n
								mySpace = LineSpace
							ENDIF ;/SearchBag[0]
						ENDIF ;/myLineValid
					ENDLOOP ;/myLine loop

					IF (myFound > 0) THEN
						Dest 	= myFound
					ENDIF

				ENDIF ;/Dest = 0

			ENDIF ;/Area Valid
			EXITIF (Dest <> 0)
		ENDLOOP ;/Area Loop
		IF (Dest <> 0) AND (Line[Dest].Space > 0) THEN
			Bag[BufferBag].Dst = USINT(Dest)
		ELSE IF (Dest <> 0) THEN
		;	Alarm[mySeq].Name = almDestinationNotValid
		ENDIF

	ELSE;//End Std.AutoAllocation
		LineSearch[1]   = D[3000 + Bag[BufferBag].Prg]
		LineSearch[2]   = D[3100 + Bag[BufferBag].Prg]
		LineSearch[3]   = D[3200 + Bag[BufferBag].Prg]
		LineSearch[4]   = D[3300 + Bag[BufferBag].Prg]
		;Check line choice 1st to 4th in order if any valid then exit loop
		LOOP Choice = 1 TO 4 DO
			LineValid = (D[100 + LineSearch[Choice]] > 0)
			LineClear = Line[LineSearch[Choice]].Clear AND (Bag[Line[LineSearch[Choice]].LastBag].Cat = 0) AND (Line[LineSearch[Choice]].SpaceBIT > 0)
			IF (LineSearch[Choice] > 0) AND LineValid AND LineClear THEN
				Bag[BufferBag].Dst = USINT(LineSearch[Choice])
			ENDIF
			EXITIF (Bag[BufferBag].Dst <> 0)
		ENDLOOP
	ENDIF ;/BufferDst > 0

ENDIF ;/BagSettled

END_PROGRAM
```

#### zzPrimSearch.var - Local variables
```iecst
(********************************************************************
 * COPYRIGHT -- HP
 ********************************************************************
 * Program: zzPrimSearch
 * File: zzPrimSearch.var
 * Author: treamsbottom
 * Created: May 09, 2014
 ********************************************************************
 * Local variables of program zzPrimSearch
 ********************************************************************)
VAR
	MaxBuffers : UINT;
	BufferBagNum : ARRAY[0..3] OF UINT;
	Buffer : UINT;
	TestBuffer : UINT;
	BufferBag : UINT;
	BufferSettled : BOOL;
	SettledBuffer : ARRAY[0..3] OF BOOL;
	BufferPrg : USINT;
	BufferCat : UDINT;
	BufferCus : UDINT;
	BufferDst : USINT;
	n : UINT;
	MinLine : UINT;
	MaxLine : UINT;
	Dest : UINT;
	Buff : UINT;
	mySeq : UINT;
	AreaChoice : ARRAY[0..4] OF UINT;
	Area : UINT;
	AreaStartLine : UINT;
	AreaEndLine : UINT;
	AreaValid : BOOL;
	myLine : UINT;
	myLineValid : BOOL;
	myLineUsed : BOOL;
	myStartStop : UINT;
	SearchBag : ARRAY[0..4] OF UINT;
	myDepth : UINT;
	MaxDepth : UINT;
	FoundDepth : UINT;
	mySpace : UINT;
	myFound : UINT;
	LineSearch : ARRAY[0..4] OF UINT;
	Choice : USINT;
	LineValid : BOOL;
	LineClear : BOOL;
	TransitBag : UINT;
	t : UINT;
	Debug : BOOL;
	Match : BOOL;
	LineSpace : UINT;
	LineIndex : USINT;
	Condtion : ARRAY[0..3] OF BOOL;
	myTransitLine : UINT;
	SearchDest : UINT;
	myBag : UINT;
	OngoingEnabled : BOOL;
END_VAR
```

### Program Logical/Sequences/10ms/zzStnSer (IEC)

#### zzstnser.var
```iecst
VAR
	MixProgTyp : BOOL;
	BatchFound : BOOL;
	MixCusts : BOOL;
	MixProgs : BOOL;
	MatchCust : BOOL;
	MatchBags : BOOL;
	MatchProgType : BOOL;
	MatchProg : BOOL;
	MatchCat : BOOL;
	StartPurge : BOOL;
	MixCats : BOOL;
	BankValid : BOOL;
	LineValid : BOOL;
	BagInList : ARRAY[0..30] OF BOOL;
	StartPurgeET : UDINT;
	BagNum : UINT;
	BagWgt : UINT;
	Index : UINT;
	PurgeBagsQty : UINT;
	StnNum : UINT;
	BatchCount : UINT;
	s : UINT;
	BatchWeight : UINT;
	myBag : UINT;
	r : UINT;
	MaxReverseWeight : UINT;
END_VAR
VAR RETAIN
	LineSearchManual : UINT;
END_VAR
VAR
	NumberOfPurgeBags : UINT;
	x : UINT;
END_VAR
VAR RETAIN
	SearchLine : UINT;
END_VAR
VAR
	Bank : UINT;
	Choice : UINT;
	EndofBagArray : UINT;
	PurgeBatchSize : UINT;
	MaxBatchWieght : UINT;
END_VAR
VAR RETAIN
	n : UINT;
END_VAR
VAR
	t : UINT;
	myBag_x : UINT;
	myBag_n : UINT;
END_VAR
VAR RETAIN
	SearchFound : UINT;
END_VAR
VAR
	LineSearch : ARRAY[0..4] OF UINT;
	SearchBagArray : ARRAY[0..30] OF UINT;
	PurgeBags : ARRAY[0..30] OF UINT;
	PurgeBagsInWgtOrder : ARRAY[0..30] OF USINT;
	PurgeOn : UINT;
	StatusReg : UDINT;
	SearchIndex : USINT;
	ReSearch : BOOL;
	MisMatchedLoad : BOOL;
	y : INT;
	Break : BOOL;
	StnCat : UDINT;
	GetStn : UINT;
	TestTim : BOOL;
	NO : BOOL;
	CHECK : UINT;
END_VAR
```

#### zzstnser.ab
```automation-basic
;-----------------------------------------------------
;Sorting Station Search Routine - No changes required!
;-----------------------------------------------------

;----------------------------------------
;Version 1.00 19/12/2005 First Issue D.J.
;Version 2.00 03/11/2010 Revised D.J.
;----------------------------------------

PROGRAM _CYCLIC

;Only one Bank / Loading VC can search in a given scan.

Bank = Bank + 1
IF (Bank > Std.MaxStationBanks) THEN
	Bank = 1
ENDIF

;Clear Array
Std.StnsToPurge = FALSE
LOOP n = 0 TO Std.MaxWeighstations DO
	;IF Stn[n].Purge THEN
	;	Std.StnsToPurge = TRUE
	;ENDIF
	BagInList[n] = FALSE
	SearchBagArray[n] = 0
ENDLOOP
TON_10ms(Std.StnsToPurge,100,StartPurge,StartPurgeET) ; use a timer to wait for all purge events to be recieved from trackview

MixCats			= (D[369] > 0)
MixCusts		= (D[366] > 0)	;Allow mixing of customers?
MixProgs		= (D[367] > 0)	;Allow mixing of Programs?

IF MixProgs	 THEN					;IF mixing programs then type must be mixed also.....
	D[368] =  1
ENDIF
MixProgTyp			= (D[368] > 0) 	;Allow mixing of Program Types?

;IF Std.ReversingBelt THEN
;	MaxReverseWeight	= D[370]			;Max weight to reverse..
;ELSE
	;MaxReverseWeight = 0
;ENDIF
;Send Status to Trackview -- BitWise OR to look at all banks

;PurgeOn = (Std.PurgeBank[1].PurgeOn OR Std.PurgeBank[2].PurgeOn OR Std.PurgeBank[3].PurgeOn OR Std.PurgeBank[4].PurgeOn)
;StatusReg = (Std.PurgeBank[1].StationsStatus OR Std.PurgeBank[2].StationsStatus OR Std.PurgeBank[3].StationsStatus OR Std.PurgeBank[4].StationsStatus)
D[360] = PurgeOn
memcpy(ADR(D[371]),ADR(StatusReg),4)
;Used by other sequences that need to check for Line[x].SpaceBIT direct
;eg. Loading VC will look for Enable.Search = 3
Enable.Search = Bank

IF (Bank <= Std.MaxStationBanks) THEN

	IF (Ldg[Bank].Search = 1) THEN

		Ldg[Bank].Found = 0
		Ldg[Bank].Line  = 0

		SearchFound = 0
		SearchLine  = 0

		Stn[0].QTime = 0
;	LOOP x = 1 TO 1 DO
		LOOP x = Ldg[Bank].StartStn TO Ldg[Bank].EndStn DO
		;	x = 11
			n = x
			;Std.StnsToPurge = TRUE    ;KEV

			IF (Std.StnsToPurge AND Std.Purging) THEN	;Search through purge Stations to find bags that can be mixed

				IF Bank = 1 THEN
					Break
;					IF NOT TestTim THEN
;						GOTO Debug
;					ENDIF
				ELSE IF Bank = 2 THEN
					Break
				ENDIF
				;Purge doesn;t need to be in x loop so exit if > 1
				EXITIF x > Ldg[Bank].StartStn
				IF StartPurge THEN
					PurgeBatchSize	= 0
					BatchFound = FALSE
					; 1st put all bags to be searched into an array to reduce scanning through all stations bags
					LOOP r = 0 TO Std.MaxWeighstations DO
				;		Std.PurgeBank[Bank].PurgeBatch[r] = 0
					;	IF Stn[r].Purge AND (Stn[r].Weight > 0) AND NOT BagInList[r] AND (r >= Ldg[Bank].StartStn) AND (r <= Ldg[Bank].EndStn)  THEN
				;			SearchBagArray[Std.MaxWeighstations] = Std.StationBagsStart[Bank] + (r-Ldg[Bank].StartStn)
				;			BagInList[r] = TRUE
					;	ENDIF
						;Shuffle array
						LOOP s = Std.MaxWeighstations DOWNTO 1 DO
							IF (SearchBagArray[s-1] = 0) AND (SearchBagArray[s] > 0) THEN
								SearchBagArray[s-1] = SearchBagArray[s]
								SearchBagArray[s] = 0
								EndofBagArray = (s - 1)
							ENDIF
						ENDLOOP
					ENDLOOP
					;LOOP r = 0 TO EndofBagArray DO ; Start Searching through bags
					r = 0 ;Only search through from 1st bag in array as we already know it is to purge
					ReSearch = FALSE
					MisMatchedLoad = FALSE
					SearchIndex = 0
					StartSearch: ;Marker to re-search
					IF ReSearch THEN
						r = SearchIndex
					ENDIF
					LOOP s = 0 TO Std.MaxWeighstations DO
						PurgeBags[s] = 0
					ENDLOOP
					LOOP s = EndofBagArray DOWNTO 0 DO
						myBag_n = SearchBagArray[r]
						myBag_x = SearchBagArray[s]
						MatchCust = FALSE
						MatchCat = FALSE
						MatchProgType = FALSE
						MatchProg = FALSE
						BankValid = TRUE;((myBag_n >= Ldg[Bank].StartStn) AND (myBag_n <= Ldg[Bank].EndStn) AND (myBag_x >= Ldg[Bank].StartStn) AND (myBag_x <= Ldg[0].EndStn))

						;Check customer 1st
						IF (Bag[myBag_n].Cus = Bag[myBag_x].Cus) OR MixCusts THEN
							MatchCust = TRUE
						ENDIF
						IF (Bag[myBag_n].Cat = Bag[myBag_x].Cat) OR MixCats	 THEN
							MatchCat = TRUE
						ENDIF
					;	IF (Bag[myBag_n].Prg = Bag[myBag_x].Prg) OR MixProgs THEN
					;		MatchProg = TRUE
					;	ENDIF
					;	IF (D[2900 + Bag[myBag_n].Prg] = D[2900 + Bag[myBag_x].Prg]) OR MixProgTyp THEN
					;		MatchProgType = TRUE
					;	ENDIF

						MatchBags = (MatchCust AND MatchCat AND MatchProg AND MatchProgType AND BankValid)
						IF MatchBags THEN ; Put bag into another array so they can be best matched by weight
							;PurgeBags[0] = myBag_n
							PurgeBags[Std.MaxWeighstations] = myBag_x
							LOOP t = Std.MaxWeighstations DOWNTO 1 DO
								IF (PurgeBags[t] > 0) AND (PurgeBags[t-1] = 0) THEN
									PurgeBags[t -1] = PurgeBags[t]
									PurgeBags[t] = 0
									PurgeBatchSize	= t
								ENDIF
							ENDLOOP
						ENDIF
					ENDLOOP ; Ony research if no matching bags, and the bag searched is to small for a batch
					IF ((PurgeBatchSize = 1) AND (Bag[PurgeBags[0]].Wgt < MaxReverseWeight)) THEN
						ReSearch = TRUE
						INC SearchIndex
						;Check when all bags have been searched...
						IF (SearchBagArray[SearchIndex] = 0) THEN
							;INC SearchIndex
							;The only bags left cannot be put in the same bag and should be classified as a mixed load.
							MisMatchedLoad = (SearchIndex > 1)
							LOOP y = 0 TO SearchIndex - 1 DO
								PurgeBags[y] = 	SearchBagArray[y]
							ENDLOOP
							PurgeBatchSize = SearchIndex
						ELSE
							GOTO StartSearch
						ENDIF
					ENDIF

					;ENDLOOP
					;Matching bags are in the array Purge Bags. Try to fit into a load?
					;Bag 0 in the array is that master.. This is the data that will go into a bag.. so we will get the batch weight from this program code.
					;Put all bag into wieght order highest first..
					LOOP r = 0 TO 19 DO
						BagInList[r] = FALSE
						PurgeBagsInWgtOrder[r] = 0
					ENDLOOP
					IF (PurgeBatchSize > 0) THEN
						GetStn =  ((PurgeBags[0] - Std.StationBagsStart[Bank]) + 1)
						IF (GetStn < Std.MaxWeighstations) THEN
							MaxBatchWieght = D[4900 + GetStn] ;SP3
						ENDIF
						IF (MaxBatchWieght = 0) OR (MaxBatchWieght <= MaxReverseWeight) THEN
							 MaxBatchWieght = MaxReverseWeight + 100
						ENDIF

						LOOP r = 0 TO (PurgeBatchSize - 1) DO
							BagWgt = 0
							LOOP s = 0 TO (PurgeBatchSize - 1) DO
								IF (Bag[PurgeBags[s]].Wgt > 0) AND (Bag[PurgeBags[s]].Wgt > BagWgt) AND NOT BagInList[s] THEN
									BagWgt = Bag[PurgeBags[s]].Wgt
									BagNum = PurgeBags[s]
									Index = s
								ENDIF
							ENDLOOP
							PurgeBagsInWgtOrder[r] = USINT(BagNum)
							BagInList[Index] = TRUE
						ENDLOOP ;
						IF (MaxBatchWieght > MaxReverseWeight) AND (Bag[PurgeBagsInWgtOrder[0]].Wgt > 0)THEN ; Check no errors in batch sizes.. Reverse all loads if fault
							;Now bags are in weight order make the best by adding the highest values until bag is full
							BatchWeight = 0
							PurgeBagsQty = 0
							;IF (Bag[PurgeBagsInWgtOrder[0]].Wgt  < MaxBatchWieght) THEN
							BatchWeight = Bag[PurgeBagsInWgtOrder[0]].Wgt
							BatchCount = Bag[PurgeBagsInWgtOrder[0]].Cnt
						;	Std.PurgeBank[Bank].PurgeBatch[0] = PurgeBagsInWgtOrder[0]
							;ENDIF
							LOOP r = 1 TO PurgeBatchSize DO ; Start from 1 as index 0 is highest weight so always in the array
								myBag = PurgeBagsInWgtOrder[r]
								IF ((Bag[myBag].Wgt + BatchWeight) <= MaxBatchWieght) THEN
									BatchWeight = Bag[myBag].Wgt + BatchWeight
									BatchCount = Bag[myBag].Cnt + BatchCount
							;		Std.PurgeBank[Bank].PurgeBatch[PurgeBatchSize] = USINT(myBag)
									PurgeBagsQty = PurgeBagsQty + 1
								ENDIF
								;Shuffle down array
								LOOP s = PurgeBatchSize DOWNTO 1 DO
								;	IF (Std.PurgeBank[Bank].PurgeBatch[s] > 0) AND (Std.PurgeBank[Bank].PurgeBatch[s - 1] = 0) THEN
								;		Std.PurgeBank[Bank].PurgeBatch[s - 1] = Std.PurgeBank[Bank].PurgeBatch[s]
								;		Std.PurgeBank[Bank].PurgeBatch[s] = 0
								;	ENDIF
								ENDLOOP
							;	IF (r = PurgeBatchSize) AND (Std.PurgeBank[Bank].PurgeBatch[0] > 0) THEN
							;		BatchFound = TRUE
							;	ENDIF
							EXITIF BatchFound = TRUE
							ENDLOOP
						ENDIF
;					ELSE
;						GOTO ExitPurge ;Invalid purge..
					ENDIF
					IF BatchFound AND NOT MisMatchedLoad THEN ;Bags found;
						IF (BatchWeight >=  MaxReverseWeight) THEN ; Wieght it OK purge into Bag search for destination.

							IF NO THEN
								SearchFound  		= 99
								SearchLine   		= 0;LineSearch[Choice]
								Ldg[Bank].Search   	= 2
							ELSE	;
								;Check line choice 1st to 4th in order if any valid then exit loop
								;StnNum = (Std.PurgeBank[Bank].PurgeBatch[0] - (Std.StationBagsStart[Bank] - Ldg[Bank].StartStn)) ; Get station number from Bag number.
						;		StnCat =  Bag[Std.PurgeBank[Bank].PurgeBatch[0]].Prg

								LineSearch[1]   = D[3000 + StnCat]
								LineSearch[2]   = D[3100 + StnCat]
								LineSearch[3]   = D[3200 + StnCat]
								LineSearch[4]   = D[3300 + StnCat]

								LOOP Choice = 1 TO 4 DO
									LineValid = (D[20 + LineSearch[Choice]] > 0)
									IF (LineSearch[Choice] > 0) AND (Line[LineSearch[Choice]].SpaceBIT >= 1) AND LineValid THEN
										SearchFound  		= 99
										SearchLine   		= LineSearch[Choice]
										Ldg[Bank].Search   	= 2
									ENDIF
									EXITIF (SearchFound > 0)
								ENDLOOP
							ENDIF
						ELSE ; Load/s is to small reverse.

							SearchFound  		= 98
							SearchLine   		= 0
							Ldg[Bank].Search   	= 2
						ENDIF
					ELSE IF MisMatchedLoad THEN
						SearchFound  		= 97
						SearchLine   		= 0
						Ldg[Bank].Search   	= 2
					ENDIF
					IF SearchFound > 90 THEN ;If bags are found remove from purging Q
;						Std.PurgeBank[Bank].PurgeBagQty	= PurgeBagsQty

;						Std.PurgeBank[Bank].PurgeBatchWieght = BatchWeight
;					Std.PurgeBank[Bank].PurgeBatchCount	= BatchCount
;						LOOP r = 0 TO PurgeBagsQty - 1 DO
;							IF (Std.PurgeBank[Bank].PurgeBatch[r] > 0) THEN
;								StnNum = (Std.PurgeBank[Bank].PurgeBatch[r] - (Std.StationBagsStart[Bank] - Ldg[Bank].StartStn))
;								;Stn[StnNum].QTime = 0
;								;Stn[StnNum].Purge = FALSE
;							ENDIF
;						ENDLOOP
					ENDIF
				ENDIF
			ELSE IF ((Stn[n].QTime > 10) AND (Stn[n].QTime > Stn[0].QTime)) THEN

				;Destination has been given to bag by operator check
				LineSearchManual = Stn[n].DestManual

				IF Std.AutoLineAllocation THEN

					;Automatic Line Allocation - Line Space is never checked even if a destiantion has been edited
					SearchFound  		= n
					SearchLine   		= LineSearchManual
					Stn[0].QTime 		= Stn[n].QTime
					Ldg[Bank].Search   	= 2

				ELSE
					;1st 2nd 3rd and 4th Line choices
					LineSearch[1]   = D[3000 + n]
					LineSearch[2]   = D[3100 + n]
					LineSearch[3]   = D[3200 + n]
					LineSearch[4]   = D[3300 + n]

					;Always Search for at least 1 space
					IF (Stn[n].SpacesRequired = 0) THEN
						Stn[n].SpacesRequired = 1
					ENDIF

					;When manual is selected then the 1st 2nd 3rd and 4th are not checked
					IF (LineSearchManual > 0) THEN
						IF (Line[LineSearchManual].SpaceBIT > 0) THEN
							SearchFound  		= n
							SearchLine   		= LineSearchManual
							Stn[0].QTime 		= Stn[n].QTime
							Ldg[Bank].Search   	= 2
						ENDIF
					ELSE
							;Check line choice 1st to 4th in order if any valid then exit loop

						LOOP Choice = 1 TO 4 DO
							;Choice = 1
							LineValid = (D[20 + LineSearch[Choice]] > 0)
							IF (LineSearch[Choice] > 0) AND (Line[LineSearch[Choice]].SpaceBIT >= Stn[n].SpacesRequired)  THEN
								SearchFound  		= n
								SearchLine   		= LineSearch[Choice]
								CHECK              =  LineSearch[Choice]
								Stn[0].QTime 		= Stn[n].QTime
								Ldg[Bank].Search   	= 2

							ENDIF
							EXITIF (SearchFound > 0)
						ENDLOOP

					ENDIF

				ENDIF ;/AutoLineAllocation

			ENDIF

		ENDLOOP

		ExitPurge:
		IF (Ldg[Bank].Search = 2) THEN
			Ldg[Bank].Found  = SearchFound
			Ldg[Bank].Line   = SearchLine
		ELSE
			Ldg[Bank].Search = 0 ;Failed
		ENDIF

	ENDIF
ENDIF
Debug:

END_PROGRAM
```

### Program Logical/Sequences/10ms/zzCount (IEC) - Counting frames inputs & Piece Weights

#### zzcount.var
```iecst
VAR
	CountPLS : ARRAY[0..49] OF R_TRIG;
	CountMode : UINT;
	CountPiece : BOOL;
	CountBoth : BOOL;
	CountCount : BOOL;
	StnUsePiece : BOOL;
	StnCountPiece : BOOL;
	StnCat : UDINT;
	CountOn : BOOL;
	StnGram : DINT;
	StnPieceWgt : UINT;
	Remainder : INT;
	Items : DINT;
	ItemsRound : DINT;
	n : UINT := 0;
END_VAR
```

### Program Logical/Sequences/10ms/zzStnMix (IEC) - * Station mixing Customer and Categories

#### zzstnmix.var
```iecst
VAR
	n	:UINT;
	CatChanged	:BOOL;
	CatValid	:BOOL;
	CusChanged	:BOOL;
	CusValid	:BOOL;
	WgtValue	:INT;
	WgtValid	:BOOL;
	StnBag	:UINT;
	CntValue	:INT;
	CntValid	:BOOL;
END_VAR
```

### Program Logical/Sequences/10ms/zzStatus (IEC) - * System status

#### zzstatus.var
```iecst
VAR
	OngoingStopped : BOOL;
	OffgoingStopped : BOOL;
	LoadingStopped : BOOL;
	tmrForce : TON_10ms;
	ForceEnable : BOOL;
	tmrBeltPLS_A : TON_10ms;
	A_PT : UDINT;
	tmrBeltPLS_B : TON_10ms;
	B_PT : UDINT;
	CarouselPhotocell : BOOL;
	tmrCaroPhotoClear : TON_10ms;
	CaroClearPT : UDINT;
	RunSB10 : BOOL;
	tmrCaroPhotoBlocked : TON_10ms;
	CaroBlockedPT : UDINT;
	tmrClearSDC3 : TON_10ms;
	SDC3BagOpen : BOOL;
	ForceBelt : BOOL;
	RunSB11 : BOOL;
	SB10Photocell : BOOL;
	SB11Photocell : BOOL;
	tmrSB11Clear : TON_10ms;
	tmrSB10Clear : TON_10ms;
	tmrBeltPLS_C : TON_10ms;
	tmrBeltPLS_D : TON_10ms;
	C_PT : UDINT;
	D_PT : UDINT;
	I_EndOfBelt : BOOL;
	O_Run : BOOL;
	I_SelectAuto : BOOL;
	n : USINT;
END_VAR
```

### Program Logical/Sequences/10ms/1_stnsa (IEC, version 1.00.0) - * Honeycombe Stations 1 - 16 - GREEN LAMPS

#### 1_stnsaCyclic.ab
```automation-basic
PROGRAM _CYCLIC
	(* cyclic program *)

;Honeycombe Sorting Station Control
;----------------------------------------------------
;Revision 1.00 10/01/2002 D.J. First Issue
;Revision 2.00 07/02/2005 D.J. Removed Stn Mix
;Revision 3.00 22/08/2006 D.J. Changed to timer array
;----------------------------------------------------

;Timers
OpenTime  = 700
CloseTime = 300

TON_10ms(    OpenBag[1],OpenTime ,BagOpened[1],BagOpenedET[1])
TON_10ms(NOT OpenBag[1],CloseTime,BagClosed[1],BagClosedET[1])
TON_10ms(    OpenBag[2],OpenTime ,BagOpened[2],BagOpenedET[2])
TON_10ms(NOT OpenBag[2],CloseTime,BagClosed[2],BagClosedET[2])
TON_10ms(    OpenBag[3],OpenTime ,BagOpened[3],BagOpenedET[3])
TON_10ms(NOT OpenBag[3],CloseTime,BagClosed[3],BagClosedET[3])
TON_10ms(    OpenBag[4],OpenTime ,BagOpened[4],BagOpenedET[4])
TON_10ms(NOT OpenBag[4],CloseTime,BagClosed[4],BagClosedET[4])
TON_10ms(    OpenBag[5],OpenTime ,BagOpened[5],BagOpenedET[5])
TON_10ms(NOT OpenBag[5],CloseTime,BagClosed[5],BagClosedET[5])
TON_10ms(    OpenBag[6],OpenTime ,BagOpened[6],BagOpenedET[6])
TON_10ms(NOT OpenBag[6],CloseTime,BagClosed[6],BagClosedET[6])
TON_10ms(    OpenBag[7],OpenTime ,BagOpened[7],BagOpenedET[7])
TON_10ms(NOT OpenBag[7],CloseTime,BagClosed[7],BagClosedET[7])
TON_10ms(    OpenBag[8],OpenTime ,BagOpened[8],BagOpenedET[8])
TON_10ms(NOT OpenBag[8],CloseTime,BagClosed[8],BagClosedET[8])
TON_10ms(    OpenBag[9],OpenTime ,BagOpened[9],BagOpenedET[9])
TON_10ms(NOT OpenBag[9],CloseTime,BagClosed[9],BagClosedET[9])
TON_10ms(    OpenBag[10],OpenTime ,BagOpened[10],BagOpenedET[10])
TON_10ms(NOT OpenBag[10],CloseTime,BagClosed[10],BagClosedET[10])
TON_10ms(    OpenBag[11],OpenTime ,BagOpened[11],BagOpenedET[11])
TON_10ms(NOT OpenBag[11],CloseTime,BagClosed[11],BagClosedET[11])
TON_10ms(    OpenBag[12],OpenTime ,BagOpened[12],BagOpenedET[12])
TON_10ms(NOT OpenBag[12],CloseTime,BagClosed[12],BagClosedET[12])
TON_10ms(    OpenBag[13],OpenTime ,BagOpened[13],BagOpenedET[13])
TON_10ms(NOT OpenBag[13],CloseTime,BagClosed[13],BagClosedET[13])
TON_10ms(    OpenBag[14],OpenTime ,BagOpened[14],BagOpenedET[14])
TON_10ms(NOT OpenBag[14],CloseTime,BagClosed[14],BagClosedET[14])
TON_10ms(    OpenBag[15],OpenTime ,BagOpened[15],BagOpenedET[15])
TON_10ms(NOT OpenBag[15],CloseTime,BagClosed[15],BagClosedET[15])
TON_10ms(    OpenBag[16],OpenTime ,BagOpened[16],BagOpenedET[16])
TON_10ms(NOT OpenBag[16],CloseTime,BagClosed[16],BagClosedET[16])

LOOP n = 1 TO Std.MaxWeighstations DO
//LOOP n = 2 TO 2 DO

	Bag[200+n].Wgt = Stn[n].Weight

	STEP = D[920 + n]
	;Setup Pulse contact
	PLS[n] = (STEP <> LASTSTEP[n])
	LASTSTEP[n] = STEP

	;Step 0 - Disabled
	IF STEP = 0 THEN
		Stn[n].LampOn = TRUE
		Stn[n].CloseFlap = TRUE
		;Disabled
	ENDIF

	IF STEP = 1 THEN
		Stn[n].LampOn = TRUE
		IF D[901] = n THEN
			D[901] = 0
		ENDIF
		IF BagClosed[n] THEN
			D[920 + n] = 2
		ENDIF
	ENDIF

	IF STEP = 2 THEN
		IF D[901] = n THEN
			D[920 + n] = 3
		ENDIF
	ENDIF

	IF STEP = 3 THEN
		Stn[n].LampOn = TRUE
		Stn[n].CloseFlap = TRUE
		;StnMix[n].Cat[0] = 0 ;Set All Mixing Registers to 0 for this station report must have been done
		IF (BagOpened[n] AND ((Stn[n].Weight < 30) OR Test.Stations) AND Ldg[1].BeltHasRun) THEN//Std.TransferBeltRun) THEN
			D[920 + n] = 1
		ENDIF
	ENDIF
	OpenBag[n] = (STEP = 3)

ENDLOOP

;Outputs
;-------

Y[12].Y05 = OpenBag[1]
Y[12].Y06 = OpenBag[2]
Y[12].Y07 = OpenBag[3]
Y[12].Y08 = OpenBag[4]
Y[13].Y05 = OpenBag[5]
Y[13].Y06 = OpenBag[6]
Y[13].Y07 = OpenBag[7]
Y[13].Y08 = OpenBag[8]
Y[14].Y05 = OpenBag[9]
Y[14].Y06 = OpenBag[10]
Y[14].Y07 = OpenBag[11]
Y[14].Y08 = OpenBag[12]
Y[15].Y05 = OpenBag[13]
Y[15].Y06 = OpenBag[14]
Y[15].Y07 = OpenBag[15]
Y[15].Y08 = OpenBag[16]

;Lamps to Outputs - From weighing / search
Y[12].Y01 = (Stn[1].LampOn  OR (Stn[1].LampFlashFast AND Std.Clock100ms) OR Stn[1].SP2 OR Stn[1].SP1 AND Std.Clock500ms)
Y[12].Y02 = (Stn[2].LampOn  OR (Stn[2].LampFlashFast AND Std.Clock100ms) OR Stn[2].SP2 OR Stn[2].SP1 AND Std.Clock500ms)
Y[12].Y03 = (Stn[3].LampOn  OR (Stn[3].LampFlashFast AND Std.Clock100ms) OR Stn[3].SP2 OR Stn[3].SP1 AND Std.Clock500ms)
Y[12].Y04 = (Stn[4].LampOn  OR (Stn[4].LampFlashFast AND Std.Clock100ms) OR Stn[4].SP2 OR Stn[4].SP1 AND Std.Clock500ms)
Y[13].Y01 = (Stn[5].LampOn  OR (Stn[5].LampFlashFast AND Std.Clock100ms) OR Stn[5].SP2 OR Stn[5].SP1 AND Std.Clock500ms)
Y[13].Y02 = (Stn[6].LampOn  OR (Stn[6].LampFlashFast AND Std.Clock100ms) OR Stn[6].SP2 OR Stn[6].SP1 AND Std.Clock500ms)
Y[13].Y03 = (Stn[7].LampOn  OR (Stn[7].LampFlashFast AND Std.Clock100ms) OR Stn[7].SP2 OR Stn[7].SP1 AND Std.Clock500ms)
Y[13].Y04 = (Stn[8].LampOn  OR (Stn[8].LampFlashFast AND Std.Clock100ms) OR Stn[8].SP2 OR Stn[8].SP1 AND Std.Clock500ms)
Y[14].Y01 = (Stn[9].LampOn  OR (Stn[9].LampFlashFast AND Std.Clock100ms) OR Stn[9].SP2 OR Stn[9].SP1 AND Std.Clock500ms)
Y[14].Y02 = (Stn[10].LampOn OR (Stn[10].LampFlashFast AND Std.Clock100ms) OR Stn[10].SP2 OR Stn[10].SP1 AND Std.Clock500ms)
Y[14].Y03 = (Stn[11].LampOn OR (Stn[11].LampFlashFast AND Std.Clock100ms) OR Stn[11].SP2 OR Stn[11].SP1 AND Std.Clock500ms)
Y[14].Y04 = (Stn[12].LampOn OR (Stn[12].LampFlashFast AND Std.Clock100ms) OR Stn[12].SP2 OR Stn[12].SP1 AND Std.Clock500ms)
Y[15].Y01 = (Stn[13].LampOn OR (Stn[13].LampFlashFast AND Std.Clock100ms) OR Stn[13].SP2 OR Stn[13].SP1 AND Std.Clock1s )
Y[15].Y02 = (Stn[14].LampOn OR (Stn[14].LampFlashFast AND Std.Clock100ms) OR Stn[14].SP2 OR Stn[14].SP1 AND Std.Clock500ms)
Y[15].Y03 = (Stn[15].LampOn OR (Stn[15].LampFlashFast AND Std.Clock100ms) OR Stn[15].SP2 OR Stn[15].SP1 AND Std.Clock500ms)
Y[15].Y04 = (Stn[16].LampOn OR (Stn[16].LampFlashFast AND Std.Clock100ms) OR Stn[16].SP2 OR Stn[16].SP1 AND Std.Clock500ms)

Y[8].Y01 = Stn[1].CloseFlap
Y[8].Y02 = Stn[2].CloseFlap
Y[8].Y03 = Stn[3].CloseFlap
Y[8].Y04 = Stn[4].CloseFlap
Y[8].Y05 = Stn[5].CloseFlap
Y[8].Y06 = Stn[6].CloseFlap
Y[8].Y07 = Stn[7].CloseFlap
Y[8].Y08 = Stn[8].CloseFlap
Y[8].Y09 = Stn[9].CloseFlap
Y[8].Y10 = Stn[10].CloseFlap
Y[8].Y11 = Stn[11].CloseFlap
Y[8].Y12 = Stn[12].CloseFlap
Y[8].Y13 = Stn[13].CloseFlap
Y[8].Y14 = Stn[14].CloseFlap
Y[8].Y15 = Stn[15].CloseFlap
Y[8].Y16 = Stn[16].CloseFlap
END_PROGRAM
```

### Program Logical/Sequences/10ms/2_belt1 (IEC) - * STB1 Transfer Belt 1

#### 2_belt1Init.ab
```automation-basic
PROGRAM _INIT
	(* init program *)
END_PROGRAM
```

#### 2_belt1Cyclic.ab
```automation-basic
PROGRAM _CYCLIC
 	(* cyclic program *)

;Sequence 2 - Transfer Belt 1 from Stations 1-12

;-----------------------------------------
;Revision 1.00 18/01/2006 D.J. First Issue
;-----------------------------------------

;Inputs and Outputs
;------------------

Bank 						= 1

I_PhotoBottom 				= X[5].X14
I_PhotoTop   				= X[5].X14

Request.TransferBelt	= FALSE

O_RunBelt 					= FALSE

Alarm[2].Name 				= 0
Alarm[2].Bag				= 220
Alarm[2].Beacon				= TRUE
Alarm[2].Extra				= 0
Alarm[2].Time				= 5000

n = D[901] ;Selected Station

STEP = D[902]
;Setup Pulse contact
PLS = (STEP <> LASTSTEP)
LASTSTEP = STEP

;Step 0 - Disabled
IF STEP = 0 THEN
	;Disabled
ENDIF

IF (D[902] > 10) THEN
	D[902] = 1
ENDIF

;Step 1 - Check no stations are releasing
IF STEP = 1 THEN
	;Don't allow stations to release
	Ldg[Bank].EnableStnRelease = FALSE
	;No Station Releaseng and switched on
	IF ((D[901] = 0) AND (D[11] > 0)) THEN
		IF (Bag[200].Cat = 0) THEN
			D[902] = 2 ;No Bag on belt
		ELSE
			D[902] = 4 ;Bag on belt
		ENDIF
	ENDIF
	Alarm[2].Name = almNoAlarm
ENDIF

;Step 2 - Enable Station search
IF STEP = 2 THEN

	;Check each station to see if a manual destination has been set
	LOOP n = Ldg[Bank].StartStn TO Ldg[Bank].EndStn DO

		StnBag = n + (Std.StationBagsStart[Bank] - 1)

		IF ((Bag[StnBag].Dst > 0) AND (Bag[StnBag].Dst < 99) AND (D[11] > 0)) THEN ;Dest 99 = Empty Bag in station
			Stn[n].DestManual = Bag[StnBag].Dst
		ELSE
			Stn[n].DestManual = 0
		ENDIF
		;For pairing set number of spaces to search for
		Stn[n].SpacesRequired = 0 ;D[2000 + Bag[StnBag].Prg]

	ENDLOOP

	;Station Search
	IF ((Ldg[Bank].Search = 0) AND (D[11] > 0) AND NOT Std.EStop) THEN
		Ldg[Bank].Search = 1
	ELSE IF ((Ldg[Bank].Search = 2) AND (Ldg[Bank].Found > 0))  THEN

		D[901] 	= Ldg[Bank].Found
		n 		= D[901]

		StnBag 	= n + (Std.StationBagsStart[Bank] - 1)

		;Clear the release button count if used
		Stn[n].ManualRelease 	= FALSE
		Stn[n].PBCount 			= 0

		;------Write Report------
		IF Std.StationReports  THEN

			IF (ReportLoading[n].Cat = 0) THEN

				;Check if anything has been added and current weight is not less than the previous
				WeightValue = Stn[n].Weight - INT(StnPrev[n].Wgt)
				WeightValid = (WeightValue > 0)

				;Check if anything has been added and current weight is not less than the previous
				CountValue = Stn[n].Count - INT(StnPrev[n].Cnt)
				CountValid = (CountValue > 0)

				IF (WeightValid OR CountValid) THEN

					;Ensure valid values as we report on either a weight or count change
					IF (WeightValue < 0) THEN
						WeightValue = 0
					ENDIF

					IF (CountValue < 0) THEN
						CountValue = 0
					ENDIF

		;			ReportLoading[n].Prg = Bag[StnBag].Prg 			;Program
					ReportLoading[n].Cat = Bag[StnBag].Cat			;Category
					ReportLoading[n].Cus = Bag[StnBag].Cus			;Customer
					ReportLoading[n].Wgt = UINT(WeightValue)		;Weight
					ReportLoading[n].Cnt = UINT(CountValue)			;Count
					ReportLoading[n].Stn = n         				;Station
					ReportLoading[n].Mcn = 0						;Machine
				;	ReportLoading[n].Bid = Bag[StnBag].Bid			;Batch ID
				ENDIF

			ENDIF

		ENDIF

		;Set Previous Cat and Cus to Current and Clear Weight and Count
;		StnPrev[n].Prg 	= Bag[StnBag].Prg
		StnPrev[n].Cat 	= Bag[StnBag].Cat
		StnPrev[n].Cus 	= Bag[StnBag].Cus
		StnPrev[n].Wgt 	= 0
		StnPrev[n].Cnt 	= 0
;		StnPrev[n].Bid 	= Bag[StnBag].Bid

		;Copy Station Data to Belt Bag
		Bag[200] 		= Bag[StnBag]			;Copy complete bag data
		Bag[200].Dst 	= USINT(Ldg[Bank].Line)	;Destination
		Bag[StnBag].Dst = 0 					;Reset Destination (Manual)

		;Clear Manual Release and Count
		Stn[n].ManualRelease 	= FALSE
		Stn[n].Count			= 0

		;If Stations are too close to the loading unit then jump to wait for loading unit
		;IF (n >= 1) AND (n <= 4) THEN
		;	D[902] = 6
		;ELSE
			BeltAddTime = (D[901] / 2)
			Ldg[Bank].EnableStnRelease = TRUE
			D[902] = 3
		;ENDIF

		Alarm[2].Name = almNoAlarm

	ENDIF
ELSE
	Ldg[Bank].Search  	= 0 ;Clear Search if not on step 2
ENDIF

;Step 3
;Open Bag and Release to Belt Conveyor
IF STEP = 3 THEN
;	O_RunBelt  = TRUE
;	IF (I_PhotoBottom OR I_PhotoTop	OR Test.TransferBelt) THEN
		D[902] = 4
;	ENDIF
;	Alarm[2].Name = almPhotocellNotMade
ENDIF

;Step 4 - Skipped
IF STEP = 4 THEN
	O_RunBelt = TRUE
	D[902] = 5
	Alarm[2].Name = almNoAlarm
ENDIF

;Step 5 - Run belt until top photocell is made.
IF STEP = 5 THEN
	O_RunBelt = TRUE
	IF I_PhotoTop OR Test.TransferBelt THEN
		D[902] = 6
	ENDIF
;	Alarm[2].Name = almPhotocellNotMade
ENDIF

;Step 6 - Wait for loading unit ready
TON_10ms((STEP = 6),10,RunBelt,Step6ET)
IF STEP = 6 THEN
	O_RunBelt = (NOT RunBelt AND Ldg[Bank].EnableStnRelease)
	IF Enable.TransferBelt THEN
		D[902] = 7
	ENDIF
ENDIF

;Step 7 - Run Belt until linen detected for 1 second and Station has emptied
TON_10ms(((STEP = 7) AND I_PhotoTop),100,LinenDetected,LinenDetectedET)
IF STEP = 7 THEN
	O_RunBelt = TRUE
	Ldg[Bank].EnableStnRelease = TRUE ;Enable Station to Open bags if they haven't been already
	IF (LinenDetected OR Test.TransferBelt) THEN
		D[902] = 8
	ENDIF
;	Alarm[2].Name = almPhotocellNotMade
ENDIF

;Step 8 - Run Belt until photocells clear for 5 seconds
TON_10ms(((STEP = 8) AND NOT I_PhotoBottom AND NOT I_PhotoTop AND NOT Std.EStop),500,BeltClear,BeltClearET)
IF STEP = 8 THEN
	O_RunBelt = TRUE
	IF (BeltClear AND MinBeltRun AND (D[901] = 0)) THEN
		D[902] = 9
	ENDIF
	IF NOT Std.EStop THEN
		IF I_PhotoBottom OR I_PhotoTop THEN
	;		Alarm[2].Name = almPhotocellBlocked
		ELSE IF (D[901] <> 0) THEN
	;		Alarm[2].Name = almStationNotClosed
		ELSE IF NOT MinBeltRun THEN
		;	Alarm[2].Name = almClearingBeltPleaseWait
		ENDIF
	ENDIF
ENDIF

;Note - Unitl the Station has closed the min belt run time won't start
;Note - Speed for Horozintal belt = 45m/min and Inclined 55m/min
BeltRunTime = (10 + BeltAddTime)
CTU((O_RunBelt AND Std.Clock1s AND (D[901] = 0) AND NOT Std.EStop),(STEP = 1),BeltRunTime,MinBeltRun,MinBeltRunCV)

;Step 9 - Check Stations Are Closed
IF STEP = 9 THEN
	;Move Belt bag to loading unit
	IF PLS AND ((Bag[220].Cat = 0) OR (Bag[220].Cat = Std.MaxCats)) AND (Bag[200].Cat > 0) THEN ;OCMW Special!!!!!!!!!
		Bag[220] = Bag[200]
		Bag[200] = Bag[0]
	ENDIF
	IF (D[901] = 0) THEN
		D[902] = 1
	ENDIF
;	Alarm[2].Name = almStationNotClosed
ENDIF

;Alarms
TimerAlarm.IN = NOT PLS AND (Alarm[2].Name > 0)
TimerAlarm.PT = Alarm[2].Time
TimerAlarm FUB TON_10ms()
Alarm[2].On = TimerAlarm.Q
Alarm[2].ET = TimerAlarm.ET

;Outputs
;Inform Station Sequences that the belt has been
Ldg[Bank].BeltHasRun = ((D[902] > 3) AND Ldg[Bank].EnableStnRelease)

Y[10].Y10 = O_RunBelt
END_PROGRAM
```

### Program Logical/Sequences/10ms/3_slu_1 (IEC) - * Loading unit SLU1

#### 3_slu_1Cyclic.ab
```automation-basic
PROGRAM _CYCLIC
	(* cyclic program *)

;Sequence 3 - Loading Unit D[903]

;Loading Unit
;--------------------------------------------------------
;Revision 1.00 09/01/2002 D.J. First Issue
;Revision 2.00 15/05/2002 D.J. Added Compression Cylinder
;--------------------------------------------------------

;I_BagAtBuffer			= X712
I_BagSLU1Trip			= X[5].X13
I_BaginLoadingUnit		= X[5].X12
;I_BagOutSLU1			= X714

I_CompressorAtTop		= X[7].X05
I_CompressorAtMid		= X[7].X06
I_CompressorAtBot		= X[7].X07
I_ChuteBlocked			= X[7].X08

O_SteadyCylinders		= FALSE
O_OpenStop	 			= FALSE
O_OpenBuffer 			= FALSE
O_BagSupport			= FALSE
O_Compression			= FALSE

Enable.SVC2				= FALSE
Alarm[3].Name 		= 0
Alarm[3].Bag		= 220
Alarm[3].Beacon		= TRUE
Alarm[3].Extra	 	= 0
Alarm[3].Time		= 3000

;Setup Sequence
;-----------------------
STEP = D[903]
;Setup Pulse contact
PLS = (STEP <> LASTSTEP)
LASTSTEP = STEP

;Alarm
;TON_10ms(((NOT PLS) AND ((STEP = 3) OR (STEP = 8) OR (STEP = 13))),3000,Alarm[3],AlarmET[3])

;Skipped - Normally Wait for Empty bag at buffer
TON_10ms((NOT I_BagSLU1Trip AND NOT I_BaginLoadingUnit),200,TripsClear,TripsClearET)
IF (STEP = 1) THEN
	IF TripsClear THEN
		D[903] = 2
	ENDIF
ENDIF

;Open stops let bag in Loading Unit
IF (STEP = 2) THEN
	O_OpenStop = TRUE
	IF I_BagSLU1Trip THEN ;bag past stop
		D[903] = 3
	ENDIF
ENDIF

Enable.SVC2 = ((STEP = 2) OR (STEP = 3)) ;Bag must be fully in loading unit before SVC2 can go back up hence STEP = 3

;Wait for bag to settle
TON_10ms(I_BaginLoadingUnit,700,EBagSettled,EBagSettledET)
IF (STEP = 3) THEN
	IF EBagSettled THEN
		D[903] = 4
	ENDIF
	Alarm[3].Name 		= almBagNotArrived
ENDIF

;Move Steady Cylinders down
TON_10ms((STEP = 4),300,SCylindersDown,SCylindersDownET)
IF (STEP = 4) THEN
	O_SteadyCylinders 	= TRUE
	O_BagSupport		= TRUE
	IF SCylindersDown THEN
		D[903] = 5
	ENDIF
ENDIF

;Wait for bag to be loaded
IF (STEP = 5) THEN
	O_SteadyCylinders 	= TRUE
	O_BagSupport		= TRUE
	IF I_CompressorAtTop THEN
		Enable.TransferBelt = TRUE
	ENDIF
	IF (Bag[220].Cat > 0) THEN
		IF I_ChuteBlocked THEN
			D[903] = 10				;If the Chute is blocked then go to service routine
		ELSE
			D[903] = 6				;Chute is clear
		ENDIF
	ENDIF
ELSE
	Enable.TransferBelt = FALSE
ENDIF

;Allow Steady Cylinders to move up
TON_10ms((STEP = 6),300,BagSupportDown,BagSupportDownET)
IF (STEP = 6) THEN
	IF BagSupportDown THEN
		D[903] = 7
	ENDIF
ENDIF

;Check svc1 is ready for a bag - If chute is blocked then goto step 10
IF (STEP = 7) THEN
	IF Enable.SLU1 THEN
		D[903] = 8
	ENDIF
ENDIF

;Open stop - unitl bag out
IF (STEP = 8) THEN
	 IF (Bag[220].Cat>0)AND(Bag[221].Cat=0) THEN
						Bag[221] = Bag[220]
						Bag[220] = Bag[0]
		ENDIF                               ;BAGMOVE2(PLS,mem_adr_E,220,221,BagSpacing)
	O_OpenStop = TRUE
	IF NOT Enable.SLU1 THEN
		D[903] = 1
	ENDIF
	Alarm[3].Name 		= almBagNotReleased
ENDIF

;Compression Cylinder Service routine
;------------------------------------
TON_10ms((STEP = 10),300,SupportDown,SupportDownET)
IF (STEP = 10) THEN
	O_SteadyCylinders 	= TRUE
	IF SupportDown THEN
		IF NOT I_ChuteBlocked THEN
			D[903] 	= 7	;Chute is clear - goto allow steadys to go up
		ELSE
			D[903] 	= 11 ;Try unblocking chute
			Tries 	= 0
		ENDIF
	ENDIF
ENDIF

;Compress Linen
TON_10ms((STEP = 11),2000,TimedOut,TimedOutET)
IF (STEP = 11) THEN
	O_SteadyCylinders 	= TRUE
	O_Compression 		= TRUE
	IF (I_CompressorAtBot OR TimedOut) THEN
		D[903] = 12
	ENDIF
ENDIF

;Allow compression to go back up
IF (STEP = 12) THEN
	O_SteadyCylinders 	= TRUE
	IF (I_CompressorAtMid OR I_CompressorAtTop) THEN
		IF NOT I_ChuteBlocked THEN
			D[903] 	= 7 	;Chute is clear - goto allow steadys to go up
		ELSE IF (Tries < 5) THEN
			D[903] 	= 11	;Re-try
			Tries	= (Tries + 1)
		ELSE
			D[903]	= 13	;Tried 5 times wait for chute to be cleared
		ENDIF
	ENDIF
ENDIF

;Compression cylinder failed wait for manual clear
IF (STEP = 13) THEN
	O_SteadyCylinders 	= TRUE
	IF (I_CompressorAtMid OR I_CompressorAtTop) THEN
		;IF NOT I_ChuteBlocked THEN
			D[903] 	= 7 	;Chute is clear - goto allow steadys to go up
		;ENDIF
	ENDIF
ENDIF

;Alarms
TimerAlarm.IN = NOT PLS AND (Alarm[3].Name > 0) //AND (AlarmOld = Alarm[3].Name)
TimerAlarm.PT = Alarm[3].Time
TimerAlarm FUB TON_10ms()
Alarm[3].On = TimerAlarm.Q
Alarm[3].ET = TimerAlarm.ET

//AlarmOld = Alarm[4].Name ;Need to ensure alarm changes as may be multiple alarms on step

;Outputs
;-------

Y[5].Y13 = O_OpenStop
;Y711 = O_OpenBuffer
Y[5].Y12 = O_SteadyCylinders
Y[7].Y02 = O_BagSupport
Y[7].Y03 = O_Compression
END_PROGRAM
```

### Program Logical/Sequences/10ms/4_spn1 (IEC, version 1.00.0) - * Soiled Low  Ongoing Transfer Lines 1 - 6

#### 4_spn1Cyclic.ab
```automation-basic
PROGRAM _CYCLIC
; 	(* cyclic program *)

;Sequence 4 - Ongoing To Storage D[904]
N

;-----------------------------------------
;Revision 1.00 09/12/2005 D.J. First Issue
;-----------------------------------------

;Inputs
OnGoingEnable 		= ((D[14] > 0) AND NOT Std.HaltSys)

I_BagatBuffer[1]	= Request.SIC[1]
I_BagatBuffer[2]	= FALSE ;X[7].X14
I_BagatBuffer[3]	= FALSE
I_BagatBuffer[4]	= FALSE

O_Reset 		  	= FALSE
O_OpenSelect[1]		= FALSE
O_OpenSelect[2]		= FALSE
O_OpenSelect[3]		= FALSE
O_OpenSelect[4]		= FALSE
Enable.SIC[1]           = FALSE

Alarm[4].Name 		= 0
Alarm[4].Bag		= 225
Alarm[4].Beacon		= TRUE
Alarm[4].Extra	 	= 0
Alarm[4].Time		= 3000

;Setup Sequence
;--------------
STEP = D[904]
;Setup Pulse contact
PLS = (STEP <> LASTSTEP)
LASTSTEP = STEP

;Check if Recirculation bag needs a destination
;IF ((Bag[107].Cat > 0) AND (Bag[107].Dst = 0) AND (D[1005] > 0) AND (D[1005] <= 6) AND (D[1006] > 0)) THEN
;	Bag[107].Dst 	= D[1005]
;	D[1006] 		= (D[1006] - 1)
;ENDIF

;Step 0 - Disabled
IF (STEP = 0) THEN
	;Disabled
ENDIF

;Step 1 - Reset Ongoing Points
TON_10ms((STEP = 1),300,ResetPoints,ResetPointsET)
IF (STEP = 1) THEN
	Dest  	= 0
	Buff 	= 0
	O_Reset = NOT ResetPoints
	IF (ResetPoints AND OnGoingEnable) THEN
		D[904] = 2
	ENDIF
ENDIF

;Set Max Buffers to search
MaxBuffers = 1

;Bag Settles at each buffer
TON_10ms(I_BagatBuffer[1],300,SettledBuffer[1],SettledBufferET[1])
;TON_10ms(Request.SVC3HighLevel,300,SettledBuffer[2],SettledBufferET[2])

BufferBagNum[1]	= 224
;BufferBagNum[2]	= 310

;Step 2 - Search for a valid Bag at one of the buffers
;Line[12].Space = PairLoopSpace
IF (STEP = 2) THEN

	Buff 	= 0
	Dest 	= 0

	IF OnGoingEnable THEN

		Alarm[4].Name 	= almNoAlarm
		Alarm[4].Time	= 2000

		LOOP Bfr = 1 TO 1 DO

			;Set Test Value for Monitoring
			IF TestBuffer > 0 THEN
				Buffer = TestBuffer
			ELSE
				Buffer = Bfr
			ENDIF

			BufferBag		= BufferBagNum[Buffer]
			BufferSettled 	= SettledBuffer[Buffer]
			BufferCat 		= Bag[BufferBag].Cat
			BufferDst 		= Bag[BufferBag].Dst

			DestValid = ((BufferDst >= 0) AND (BufferDst <= 11))

			IF (BufferSettled AND (BufferCat > 0) AND DestValid AND (Bag[225].Cat = 0)) THEN
				n = BufferDst

				IF ((Line[n].Space > 0) AND Line[n].Clear) THEN
					Dest = n
					Buff = Buffer
					;IF (Buffer = 1) OR (Buffer = 2) THEN
						D[904] 	= 3
					;ENDIF

				ELSE
			;		Alarm[4].Name 	= almDestinationNotValid
					Alarm[4].Bag	= BufferBag
				ENDIF
			ENDIF

			;Buffer Alarms
			IF (BufferCat > 0) AND NOT BufferSettled THEN
				Alarm[4].Name 	= almBagNotAtProx
				Alarm[4].Bag	= BufferBag
			ELSE IF (BufferCat = 0) AND BufferSettled THEN
			;	Alarm[4].Name 	= almBagNotShownOnScreen
				Alarm[4].Bag	= BufferBag
			ENDIF

		ENDLOOP

	ENDIF

ENDIF

;Clear Line Selections
LOOP n = 1 TO Std.MaxLines DO
	LineSelect[n] = FALSE
ENDLOOP

;Step 3 - Enable VC1 to Release a bag
IF (STEP = 3) THEN
	;Enable.SVC[1] 		= TRUE

	;IF PLS THEN
	;	C[Dest] 	= 0
	;ENDIF

	;LineSelect[Dest] 	= TRUE
	;IF NOT Request.SVC[1] THEN
		D[904] = 4
	;ENDIF
ENDIF

;Step 4 - Select line / open buffer stop
IF (STEP = 4) THEN
	Enable.SIC[1] 		= TRUE
	LineSelect[Dest] 	= TRUE
	O_OpenSelect[Buff]    = TRUE

	IF PLS THEN
		C[Dest] = 0
		IF ((Bag[224].Cat > 0) AND (Bag[225].Cat = 0)) THEN
			Bag[225] = Bag[224]
			Bag[224] = Bag[0]
		ENDIF

	ENDIF

	;Bag arrived on selected line
	IF Line[Dest].Trip THEN
		D[498] 						= Bag[225].Cus	;Set Customer for Customer FIFO
		Bag[225].Dst 				= 0 		    ;Clear Destination
		Bag[Line[Dest].LastBag] 	= Bag[225]
		Bag[225] 					= Bag[0]
		D[904] 						= 1
	ENDIF

	Alarm[4].Name = almBagNotArrived

ENDIF

;Alarms
TimerAlarm.IN = NOT PLS AND (Alarm[4].Name > 0) AND (AlarmOld = Alarm[4].Name)
TimerAlarm.PT = Alarm[4].Time
TimerAlarm FUB TON_10ms()
Alarm[4].On = TimerAlarm.Q
Alarm[4].ET = TimerAlarm.ET

AlarmOld = Alarm[4].Name ;Need to ensure alarm changes as may be multiple alarms on step 2

;Storage Line Selections
Y[4].Y11 = Reset
Y[4].Y01 = LineSelect[1]
Y[4].Y02 = LineSelect[2]
Y[4].Y03 = LineSelect[3]
Y[4].Y04 = LineSelect[4]
Y[4].Y05 = LineSelect[5]
Y[4].Y06 = LineSelect[6]
Y[4].Y07 = LineSelect[7]
Y[4].Y08 = LineSelect[8]
Y[4].Y09 = LineSelect[9]
Y[4].Y10 = LineSelect[10]

END_PROGRAM
```

### Program Logical/Sequences/10ms/5_spf1 (IEC, version 1.00.0) - * Soiled Offgoing Transfer Lines 1 - 10

#### 5_spf1Cyclic.ab
```automation-basic
PROGRAM _CYCLIC
	(* cyclic program *)

;----------------------------------------
;Sequence 5 - SPF1 Offgoing Points D[905]
;----------------------------------------
;Inputs
;------

OffGoingEnable 		= ((D[15] > 0) AND NOT Std.HaltSys)

;I_SDCBagAtBuffer[1] = X[6].X01 ;Use for single bag buffer
;I_SDCBagAtBuffer[2] = FALSE ;X[6].X13 ;Use for single bag buffer

;O_SDCBufferOpen[1]  = Y[6].Y01 ;Use for single bag buffer
;O_SDCBufferOpen[2]  = FALSE ;Y[6].Y16 ;Use for single bag buffer

I_BagAtStop[1]  = X[4].X12
I_BagAtStop[2]  = X[4].X13
I_BagAtStop[3]  = X[4].X14
I_BagAtStop[4]  = X[4].X15
I_BagAtStop[5]  = X[4].X16
I_BagAtStop[6]  = X[5].X01
I_BagAtStop[7]  = X[5].X02
I_BagAtStop[8]  = X[5].X03
I_BagAtStop[9]  = X[5].X04
I_BagAtStop[10] = X[5].X05
I_BagAtStop[11] = X[5].X06

;I_BagReleased       = X[14].X03

O_Reset 			= FALSE

;Buffer line configuration
;-------------------------
MaxBuffers			= 2

Alarm[5].Name 		= 0
Alarm[5].Bag		= 226
Alarm[5].Beacon		= TRUE
Alarm[5].Extra	 	= 0
Alarm[5].Time		= 3000

;BufferClear[1] 		= ((D[21] > 0) AND (Bag[190].Cat = 0) AND (Line[21].SpaceBIT > 0) AND (Line[21].Clear))
;BufferClear[2]		= ((D[22] > 0) AND (Bag[190].Cat = 0) AND (Line[22].Space > 0)AND (Line[22].Clear))

Uld[1].SDCReady 	= ((D[16] = 1) AND Line[12].Clear AND NOT Y[3].Y01)
Uld[2].SDCReady 	= ((D[17] = 1) AND Line[13].Clear)
;Passed to unloading search
;Uld[3].SDCReady		= FALSE
;Uld[4].SDCReady 	= FALSE

Alarm[5].Name 		= 0
Alarm[5].Bag		= 190
Alarm[5].Beacon		= TRUE
Alarm[5].Extra		= 0
Alarm[5].Time		= 3000

;Setup Sequence
;--------------
STEP = D[905]
;Setup Pulse contact
PLS = (STEP <> LASTSTEP)
LASTSTEP = STEP

;Sequence Steps
;--------------
IF (STEP = 0) THEN
	;Disabled
ENDIF

;Step 1 - Reset Points
TON_10ms((STEP = 1),300,ResetPoints,ResetPointsET)
IF (STEP = 1) THEN
	O_Reset 	= NOT ResetPoints
	FoundLine 	= 0
	Destination = 0
	IF (ResetPoints AND OffGoingEnable) THEN
		D[905] = 2
	ENDIF
ENDIF

;Bags on storage line timers
R_TRIG(Std.Clock100ms,IncSettle)
AlarmBagNotProx 	= FALSE
AlarmBagNotProxLine = 0

LOOP n = 1 TO Std.MaxLines DO

	LineSettle[n]  = (I_BagAtStop[n] AND (Bag[Line[n].FirstBag].Cat > 0))
	IF IncSettle AND LineSettle[n] AND (BagSettledTime[n] < $FFFF) THEN
		BagSettledTime[n] = BagSettledTime[n] + 1
	ELSE IF NOT LineSettle[n] THEN
		BagSettledTime[n] = 0
		;If Bag has destiantion and not at stop then alarm
		IF (STEP = 2) AND (Bag[Line[n].FirstBag].Dst > 0) THEN
			Alarm[5].Name	= almBagNotAtProx
			Alarm[5].Bag	= Line[n].FirstBag
			Alarm[5].Extra 	= n
		ENDIF
	ENDIF

ENDLOOP

;Buffer trip not correct alarms
LOOP n = 1 TO MaxBuffers DO
	IF (STEP = 2) AND BufferClear[n] AND NOT Uld[n].SDCReady THEN
		Alarm[5].Name 	= almSwitchFault
		Alarm[5].Bag	= BufferBag[n]
	ENDIF
ENDLOOP

;Search for the bag with a valid destination that has been waiting the longest
IF STEP = 2 THEN

	FoundLine 	= 0
	Destination = 0
	BestTime 	= 0
	SettleTime = 30 ;3 seconds

	LOOP n = 1 TO Std.MaxLines DO

		IF (BagSettledTime[n] > SettleTime) THEN
			SearchDest = Bag[Line[n].FirstBag].Dst

			SDC1_Valid  = ((SearchDest = 12) AND Uld[1].SDCReady)
			SDC2_Valid 	= ((SearchDest = 13) AND Uld[2].SDCReady)
			;SDC3_Valid 	= ((SearchDest = 13) AND Uld[3].SDCReady)
			;SDC4_Valid 	= ((SearchDest = 14) AND Uld[4].SDCReady)

			IF (SDC1_Valid OR SDC2_Valid OR SDC3_Valid OR SDC4_Valid) THEN
				FoundLine 	= n
				Destination = SearchDest
				BestTime 	= BagSettledTime[n]
			ENDIF
		ENDIF

	ENDLOOP

	IF ((FoundLine > 0) AND OffGoingEnable AND (Bag[226].Cat = 0) AND Line[Destination].Clear AND (Bag[226].Cat = 0) AND NOT I_BagReleased) THEN
		C[Destination]  = 0
		D[905] = 3
	ENDIF

ENDIF

;Step 3 - Select Line / Open Stop, Until Bag at correct destination
;Clear Line Selections
LOOP n = 1 TO Std.MaxLines DO
	LineSelect[n] = FALSE
ENDLOOP

IF (STEP = 3) THEN

	;Show bag in transit
	IF (Bag[226].Cat = 0) AND (Bag[Line[FoundLine].FirstBag].Cat > 0)THEN
		Bag[226] 						= Bag[Line[FoundLine].FirstBag]
		Bag[Line[FoundLine].FirstBag] 	= Bag[0]
	ENDIF

	IF PLS THEN
			;C[13] = 0
		ENDIF

	;Select Line - Wait for bag to arrive
	LineSelect[FoundLine] = TRUE

	;Select Route
	;IF (I_BagReleased  AND (Bag[Line[13].LastBag].Cat = 0)) THEN
		 ;Unloading Program
	IF (Destination = 12) AND Line[Destination].Trip THEN
		Uld[1].DischargerStartLine = FoundLine
		Bag[227] = Bag[226]
		Bag[226] = Bag[0]
		D[905] 					= 1
	ELSE IF (Destination = 13) AND Line[Destination].Trip THEN
		Uld[2].DischargerStartLine = FoundLine
		Bag[230] = Bag[226]
		Bag[226] = Bag[0]
		D[905] 					= 1
	ENDIF

	Alarm[5].Name	= almBagNotReleased

ENDIF

;move transit bag to buffer
;IF (Bag[190].Cat > 0) AND Line[13].Trip AND (Bag[193].Cat = 0) AND NOT PLS THEN
;	Bag[193] = Bag[190]
;	Bag[190] = Bag[0]
;ENDIF

;Alarms
TimerAlarm.IN = NOT PLS AND (Alarm[5].Name > 0)
TimerAlarm.PT = Alarm[5].Time
TimerAlarm FUB TON_10ms()
Alarm[5].On = TimerAlarm.Q
Alarm[5].ET = TimerAlarm.ET

;Outputs
;-------
Y[5].Y07 = O_Reset
Y[4].Y12 = LineSelect[1]
Y[4].Y13 = LineSelect[2]
Y[4].Y14 = LineSelect[3]
Y[4].Y15 = LineSelect[4]
Y[4].Y16 = LineSelect[5]
Y[5].Y01 = LineSelect[6]
Y[5].Y02 = LineSelect[7]
Y[5].Y03 = LineSelect[8]
Y[5].Y04 = LineSelect[9]
Y[5].Y05 = LineSelect[10]
Y[5].Y06 = LineSelect[11]
;Y000 = LineSelect[12]
;Y000 = LineSelect[13]
;Y000 = LineSelect[14]

Y[5].Y09 = (D[36] = 1)
Y[5].Y08 = (D[36] = 2)

;Buffer line selection
;Y[4].Y15 = (Destination = 11)
;Y[4].Y16 = (Destination = 12)
;Y[40].Y07 = (Destination = 22)
;Y[40].Y08 = (Destination = 21)
END_PROGRAM
```

### Program Logical/Sequences/10ms/6_sdc1 (IEC, version 1.00.0) - * SDC1 Machine 1 BCD/CAN

#### 6_sdc1Cyclic.ab
```automation-basic
PROGRAM _CYCLIC
	(* cyclic program *)

;Sequence 6 - Discharger 1 D[906]
a

;-----------------------------------------
;Revision 1.00 19/12/2005 D.J. First Issue
;-----------------------------------------

DischargerEnable 		= ((D[16] > 0) AND NOT Std.HaltSys)

I_BagAtBuffer			  = X[3].X02
I_BagAtDischarger = X[3].X01
I_BagEmpty        = X[5].X11

I_OpenBag				= CAN[1].DropLoad OR TestDrop           ;X[23].X01
I_LoadDropped			= CAN[1].LoadDropped OR TestDischarger  ;X[23].X02

O_Steadys				= FALSE ;Y[6].Y01
O_OpenBuffer 			= FALSE ;Y[6].Y02
O_OpenBag				= FALSE ;Y[6].Y03
O_OpenStop				= FALSE ;Y[6].Y04
O_Closer				= FALSE ;Y[6].Y05

;Alarm
Alarm[6].Name 			= 0 ;Clear sequence alarm name
Alarm[6].Bag 			= 228
Alarm[6].Beacon			= TRUE
Alarm[6].Extra			= 0
Alarm[6].Time			= 3000

;Setup Sequence
STEP = D[906]
;Setup Pulse contact
PLS = (STEP <> LASTSTEP)
LASTSTEP = STEP

;Step 0 - Disabled
IF (STEP = 0) THEN
	;Disabled
ENDIF

;Check Status - Bag settled at buffer, no bag at discharger, bag at buffer on screen and no bag at discharger on the screen
TON_10ms(I_BagAtBuffer,300,SettledAtBuffer,SettledAtBufferET)
IF (STEP = 1) THEN
	IF (DischargerEnable AND SettledAtBuffer AND NOT I_BagAtDischarger AND (Bag[228].Cat = 0) AND NOT Std.HaltSys) THEN
		D[906] = 2
	ENDIF
	IF (Bag[228].Cat > 0) THEN
		Alarm[6].Name = almBagDataError
	ELSE IF I_BagAtDischarger THEN
		Alarm[6].Name = almSwitchFault
	ENDIF
ENDIF

;Wait for bag in discharger
IF (STEP = 2) THEN
	O_OpenBuffer 	= TRUE
	;Enable.SDC[1] 	= TRUE
	IF I_BagAtDischarger THEN
		D[906] = 3
	ENDIF
	Alarm[6].Name = almBagNotArrived
ENDIF

;Let bag settle in discharger
TON_10ms(((STEP = 3) AND I_BagAtDischarger),1000,SettledAtDischarger,SettledAtDischargerET)
IF (STEP = 3) THEN
	IF (Bag[228].Cat = 0) AND (Bag[227].Cat > 0) THEN
		Bag[228] = Bag[227]
		Bag[227] = Bag[0]
	ENDIF
	IF SettledAtDischarger THEN
		D[906] = 4
	ENDIF
	Alarm[6].Name = almBagNotSettled
ENDIF

;Allow steadys to move down
TON_10ms((STEP = 4),400,SteadysDown,SteadysDownET)
IF (STEP = 4) THEN
	IF SteadysDown AND (Bag[228].Cat <> Std.MaxCats)  THEN
		D[906] = 5
	ENDIF
	IF (Bag[228].Cat = Std.MaxCats) AND SteadysDown THEN
		D[906] = 8
	ENDIF
ENDIF

;Steady cylinders on from steps 4 - 9
O_Steadys = ((STEP >= 4) AND (STEP <= 9))

;Bag opener on from step 5 - 8
O_OpenBag = ((STEP >= 6) AND (STEP <= 8))

;Wash Codes
IF (STEP = 4) OR (STEP = 5) THEN

;round up weight to give to wash machine
	Remainder = SINT(Bag[228].Wgt MOD 10)
	IF (Remainder > 4) THEN
		WgtRound = (Bag[228].Wgt + 10)
	ELSE
		WgtRound = Bag[228].Wgt
	ENDIF

;Codes to CBW
	CAN[1].Category = Bag[228].Cat
	CAN[1].Customer = Bag[228].Cus
	CAN[1].Weight   = (WgtRound / 10)
ELSE
	CAN[1].Category = 0
	CAN[1].Customer = 0
	CAN[1].Weight   = 0
ENDIF

;Bag Ready to Washing Machine
IF (STEP = 5) THEN
	CAN[1].BagReady = TRUE
	IF I_OpenBag OR TestDischarger THEN
		D[906] = 6
	ENDIF
ELSE
	CAN[1].BagReady = FALSE
ENDIF

;Set LoadDropped to False
IF (STEP <> 6) THEN
	LoadDropped = FALSE
ENDIF

;Open Bag Until LoadDropped recieved and has been open for 6 seconds
TON_10ms((STEP = 6),600,MinOpen,MinOpenET) ;ET means Elapsed Time
IF (STEP = 6) THEN

	IF I_LoadDropped OR TestDischarger THEN
	;IF I_BagEmpty THEN
		LoadDropped = TRUE
	ENDIF

	IF (LoadDropped AND MinOpen) THEN
		;Write Report
		;------------
		IF (ReportUnloading[1].Cat = 0) THEN
			ReportUnloading[1].Cat = UINT(Bag[228].Cat)	;Category
			ReportUnloading[1].Cus = UINT(Bag[228].Cus)   ;Customer
			ReportUnloading[1].Wgt = Bag[228].Wgt		;Weight
			ReportUnloading[1].Cnt = 0					;Count
			ReportUnloading[1].Stn = 0					;Station
			ReportUnloading[1].Mcn = 1					;Machine
			;Bag[201]               = Bag[120]           ;move bag into machine tracking
		ENDIF
	ENDIF
	IF (LoadDropped AND MinOpen) THEN
		D[906] = 7
	ENDIF
	Alarm[6].Name = almLoadNotDropped
ENDIF

;Change display to empty bag
IF (STEP = 7) THEN
	IF ((NOT I_OpenBag AND NOT I_LoadDropped OR TestDrop)) THEN ;AND I_BagEmpty) OR TestDrop) THEN
		Bag[228].Cat 	= Std.MaxCats
		D[906] 			= 8
	ENDIF
	Alarm[6].Name = almGeneralSequence
ENDIF

;Close bag
TON_10ms((STEP = 8),700,CloserDown,CloserDownET)
IF (STEP = 8) THEN
	O_Closer = TRUE
	IF CloserDown THEN
		D[906] = 9
	ENDIF
ENDIF

;Allow closer to go back up
TON_10ms((STEP = 9),700,CloserUp,CloserUpET)
IF (STEP = 9) THEN
	IF CloserUp THEN
		D[906] = 10
	ENDIF
ENDIF

;Allow steadys to go up
TON_10ms((STEP = 10),400,SteadyUp,SteadyUpET)
IF (STEP = 10) THEN
	IF SteadyUp THEN
		D[906] = 11
	ENDIF
ENDIF

;Check for space on empty bag buffer
IF (STEP = 11) THEN
 Request.SDC[1] = TRUE
	IF Enable.SDC[1] THEN
		D[906] = 12
	ENDIF
	ELSE
		Request.SDC[1] = FALSE
ENDIF

;Open buffer stop - unitl bag out
IF (STEP = 12) THEN
	O_OpenStop = TRUE
	IF PLS THEN
		;C[14] = 0
	ENDIF
	Bag[228].Cat = 0
	Bag[228].Cus = 0
	Bag[228].Wgt = 0
	IF NOT Enable.SDC[1] THEN
		D[906] = 1
	ENDIF
	Alarm[6].Name = almBagNotReleased
ENDIF

;Alarms
TimerAlarm.IN 	= NOT PLS AND (Alarm[6].Name > 0)
TimerAlarm.PT 	= Alarm[6].Time
TimerAlarm FUB TON_10ms()
Alarm[6].On 	= TimerAlarm.Q
Alarm[6].ET 	= TimerAlarm.ET

;Outputs

Y[3].Y01 = O_OpenBuffer
Y[3].Y02 = O_Steadys
Y[3].Y03 = O_OpenBag
Y[3].Y04 = O_OpenStop
Y[3].Y05 = O_Closer

END_PROGRAM
```

#### 6_sdc1.var
```iecst
VAR RETAIN
	STEP : UINT;
	PLS : BOOL;
	LASTSTEP : UINT;
	SteadyUp : BOOL;
	CloserUpET : TIME;
	SteadysDown : BOOL;
	SteadysDownET : TIME;
	LoadDropped : BOOL;
END_VAR
VAR
	SteadyUpET : TIME;
	CloserDownET : TIME;
	SettledAtDischargerET : TIME;
	MinOpenET : TIME;
	SettledAtDischarger : BOOL;
	CloserDown : BOOL;
	MinOpen : BOOL;
	CloserUp : BOOL;
	SettledAtBuffer : BOOL;
	SettledAtBufferET : TIME;
	I_BagAtBuffer : BOOL;
	O_OpenStop : BOOL;
	O_OpenBag : BOOL;
	O_Steadys : BOOL;
	O_OpenBuffer : BOOL;
	O_Closer : BOOL;
	I_BagAtDischarger : BOOL;
	I_OpenBag : BOOL;
	I_LoadDropped : BOOL;
	TestDrop : BOOL;
	DischargerEnable : BOOL;
	TestDischarger : BOOL;
	Remainder : SINT;
	TimerAlarm : TON_10ms;
	WgtRound : UINT;
	a : BOOL;
	I_BagEmpty : BOOL;
END_VAR
```

### Program Logical/Sequences/10ms/7_sdc2 (IEC) - * SDC1 Machine 1 BCD/CAN

#### 6_sdc1.var
```iecst
VAR RETAIN
	STEP : UINT;
END_VAR
VAR
	PLS : BOOL;
END_VAR
VAR RETAIN
	LASTSTEP : UINT;
END_VAR
VAR
	SteadyUp : BOOL;
	CloserUpET : TIME;
	SteadysDown : BOOL;
	SteadysDownET : TIME;
	LoadDropped : BOOL;
	SteadyUpET : TIME;
	CloserDownET : TIME;
	SettledAtDischargerET : TIME;
	MinOpenET : TIME;
	SettledAtDischarger : BOOL;
	CloserDown : BOOL;
	MinOpen : BOOL;
	CloserUp : BOOL;
	SettledAtBuffer : BOOL;
	SettledAtBufferET : TIME;
	I_BagAtBuffer : BOOL;
	O_OpenStop : BOOL;
	O_OpenBag : BOOL;
	O_Steadys : BOOL;
	O_OpenBuffer : BOOL;
	O_Closer : BOOL;
	I_BagAtDischarger : BOOL;
	I_OpenBag : BOOL;
	I_LoadDropped : BOOL;
	TestDrop : BOOL;
	DischargerEnable : BOOL;
	TestDischarger : BOOL;
	Remainder : SINT;
	TimerAlarm : TON_10ms;
	WgtRound : UINT;
	a : BOOL;
	I_BagEmpty : BOOL;
END_VAR
```
